# B&R Automation Studio project HISTest (part 6)

#### PMSDataTxParsing.st
```iecst
ACTION ActPMSDATATxParshing:

	PMS.SysBatProduct.Value[0]		:= SHL(USINT_TO_DWORD(PMS.SysBatProduct.Field.BSA_Production_Num), 24) OR SHL(USINT_TO_DWORD(PMS.SysBatProduct.Field.BSA_Production_Type), 16) OR UINT_TO_DWORD(PMS.SysBatProduct.Field.BSA_Production_Year);
	PMS.SysBatProduct.Value[1]		:= SHL(USINT_TO_DWORD(PMS.SysBatProduct.Field.BSA_Production_BSA_Parallel), 16) OR SHL(USINT_TO_DWORD(PMS.SysBatProduct.Field.BSA_Production_BSA_Serial), 8) OR USINT_TO_DWORD(PMS.SysBatProduct.Field.BSA_Production_VER);

	PMS.SysBatCal.Value[0]			:= SHL(REAL_TO_DWORD(PMS.SysBatCal.Field.BSA_Curr_Total), 16) OR REAL_TO_DWORD(PMS.SysBatCal.Field.BSA_Volt_Total);
	PMS.SysBatCal.Value[1] 			:= SHL(UINT_TO_DWORD(PMS.SysBatCal.Field.BSA_Divice_Status), 16) OR REAL_TO_DWORD(PMS.SysBatCal.Field.BSA_SOC);

	PMS.SysBatPWR.Value[0]			:= SHL(REAL_TO_DWORD(PMS.SysBatPWR.Field.BSA_Peak_Charge_Power_Limit), 16) OR REAL_TO_DWORD(PMS.SysBatPWR.Field.BSA_Cont_Charge_Power_Limit);
	PMS.SysBatPWR.Value[1] 			:= SHL(REAL_TO_DWORD(PMS.SysBatPWR.Field.BSA_Peak_Discharge_Power_Limit), 16) OR REAL_TO_DWORD(PMS.SysBatPWR.Field.BSA_Cont_Discharge_Power_Limit);

	PMS.SysCellVolt.Value[0]		:= SHL(REAL_TO_DWORD(PMS.SysCellVolt.Field.BSA_Cell_MinV), 16) OR REAL_TO_DWORD(PMS.SysCellVolt.Field.BSA_Cell_MaxV);
	PMS.SysCellVolt.Value[1] 		:= SHL(REAL_TO_DWORD(PMS.SysCellVolt.Field.BSA_Cell_DeviV), 16) OR REAL_TO_DWORD(PMS.SysCellVolt.Field.BSA_Cell_AVGV);

	PMS.SysCellTemps.Value[0]		:= SHL(REAL_TO_DWORD(PMS.SysCellTemps.Field.BSA_Cell_MinT), 16) OR REAL_TO_DWORD(PMS.SysCellTemps.Field.BSA_Cell_MaxT);
	PMS.SysCellTemps.Value[1] 		:= SHL(REAL_TO_DWORD(PMS.SysCellTemps.Field.BSA_Cell_DeviT), 16) OR REAL_TO_DWORD(PMS.SysCellTemps.Field.BSA_Cell_AVGT);

	PMS.SysCellV_TPos.Value[0]		:= SHL(UINT_TO_DWORD(PMS.SysCellV_TPos.Field.BSA_Cell_MinV_Location), 24) OR SHL(UINT_TO_DWORD(PMS.SysCellV_TPos.Field.BSA_Rack_MinV_Location), 16) OR SHL(USINT_TO_DWORD(PMS.SysCellV_TPos.Field.BSA_Cell_MinV_Location), 8) OR UINT_TO_DWORD(PMS.SysCellV_TPos.Field.BSA_Rack_MaxV_Location);
	PMS.SysCellV_TPos.Value[1] 		:= SHL(UINT_TO_DWORD(PMS.SysCellV_TPos.Field.BSA_Cell_MinT_Location), 24) OR SHL(UINT_TO_DWORD(PMS.SysCellV_TPos.Field.BSA_Rack_MinT_Location), 16) OR SHL(USINT_TO_DWORD(PMS.SysCellV_TPos.Field.BSA_Cell_MinT_Location), 8) OR UINT_TO_DWORD(PMS.SysCellV_TPos.Field.BSA_Rack_MaxT_Location);

	PMS.SysBatProtect.Value[0].0	:=	PMS.SysBatProtect.Field.BSA_Alarm_OC	;
	PMS.SysBatProtect.Value[0].1	:=	PMS.SysBatProtect.Field.BSA_Alarm_SOC_OV	;
	PMS.SysBatProtect.Value[0].2	:=	PMS.SysBatProtect.Field.BSA_Alarm_SOC_UN	;
	PMS.SysBatProtect.Value[0].3	:=	PMS.SysBatProtect.Field.BSA_Alarm_OV	;
	PMS.SysBatProtect.Value[0].4	:=	PMS.SysBatProtect.Field.BSA_Alarm_UV	;
	PMS.SysBatProtect.Value[0].5	:=	PMS.SysBatProtect.Field.BSA_Alarm_Cell_OV	;
	PMS.SysBatProtect.Value[0].6	:=	PMS.SysBatProtect.Field.BSA_Alarm_Cell_UV	;
	PMS.SysBatProtect.Value[0].7	:=	PMS.SysBatProtect.Field.BSA_Alarm_Cell_UnBalaV	;
	PMS.SysBatProtect.Value[0].8	:=	PMS.SysBatProtect.Field.BSA_Alarm_Discharger_Cell_OT	;
	PMS.SysBatProtect.Value[0].9	:=	PMS.SysBatProtect.Field.BSA_Alarm_Charger_Cell_OT	;
	PMS.SysBatProtect.Value[0].10	:=	PMS.SysBatProtect.Field.BSA_Alarm_Discharger_Cell_UT	;
	PMS.SysBatProtect.Value[0].11	:=	PMS.SysBatProtect.Field.BSA_Alarm_Charger_Cell_UT	;
	PMS.SysBatProtect.Value[0].12	:=	PMS.SysBatProtect.Field.BSA_Alarm_Cell_UnBalaT	;
	PMS.SysBatProtect.Value[0].13	:=	PMS.SysBatProtect.Field.BSA_Alarm_Continuously_OP	;
	PMS.SysBatProtect.Value[0].14	:=	PMS.SysBatProtect.Field.BSA_Alarm_Peak_OP	;

	PMS.SysBatProtect.Value[0].16	:=	PMS.SysBatProtect.Field.BSA_Fault_OC	;
	PMS.SysBatProtect.Value[0].17	:=	PMS.SysBatProtect.Field.BSA_Fault_SOC_OV	;
	PMS.SysBatProtect.Value[0].18	:=	PMS.SysBatProtect.Field.BSA_Fault_SOC_UN	;
	PMS.SysBatProtect.Value[0].19	:=	PMS.SysBatProtect.Field.BSA_Fault_OV	;
	PMS.SysBatProtect.Value[0].20	:=	PMS.SysBatProtect.Field.BSA_Fault_UV	;
	PMS.SysBatProtect.Value[0].21	:=	PMS.SysBatProtect.Field.BSA_Fault_Cell_OV	;
	PMS.SysBatProtect.Value[0].22	:=	PMS.SysBatProtect.Field.BSA_Fault_Cell_UV	;
	PMS.SysBatProtect.Value[0].23	:=	PMS.SysBatProtect.Field.BSA_Fault_Cell_UnBalaV	;
	PMS.SysBatProtect.Value[0].24	:=	PMS.SysBatProtect.Field.BSA_Fault_Discharger_Cell_OT	;
	PMS.SysBatProtect.Value[0].25	:=	PMS.SysBatProtect.Field.BSA_Fault_Charger_Cell_OT	;
	PMS.SysBatProtect.Value[0].26	:=	PMS.SysBatProtect.Field.BSA_Fault_Discharger_Cell_UT	;
	PMS.SysBatProtect.Value[0].27	:=	PMS.SysBatProtect.Field.BSA_Fault_Charger_Cell_UT	;
	PMS.SysBatProtect.Value[0].28	:=	PMS.SysBatProtect.Field.BSA_Fault_Cell_UnBalaT	;
	PMS.SysBatProtect.Value[0].29	:=	PMS.SysBatProtect.Field.BSA_Fault_Continuously_OP	;
	PMS.SysBatProtect.Value[0].30	:=	PMS.SysBatProtect.Field.BSA_Fault_Peak_OP	;
	PMS.SysBatProtect.Value[1].0	:=	PMS.SysBatProtect.Field.BSA_Prtct_OC	;
	PMS.SysBatProtect.Value[1].1	:=	PMS.SysBatProtect.Field.BSA_Prtct_SOC_OV	;
	PMS.SysBatProtect.Value[1].2	:=	PMS.SysBatProtect.Field.BSA_Prtct_SOC_UN	;
	PMS.SysBatProtect.Value[1].3	:=	PMS.SysBatProtect.Field.BSA_Prtct_OV	;
	PMS.SysBatProtect.Value[1].4	:=	PMS.SysBatProtect.Field.BSA_Prtct_UV	;
	PMS.SysBatProtect.Value[1].5	:=	PMS.SysBatProtect.Field.BSA_Prtct_Cell_OV	;
	PMS.SysBatProtect.Value[1].6	:=	PMS.SysBatProtect.Field.BSA_Prtct_Cell_UV	;
	PMS.SysBatProtect.Value[1].7	:=	PMS.SysBatProtect.Field.BSA_Prtct_Cell_UnBalaV	;
	PMS.SysBatProtect.Value[1].8	:=	PMS.SysBatProtect.Field.BSA_Prtct_Discharger_Cell_OT	;
	PMS.SysBatProtect.Value[1].9	:=	PMS.SysBatProtect.Field.BSA_Prtct_Charger_Cell_OT	;
	PMS.SysBatProtect.Value[1].10	:=	PMS.SysBatProtect.Field.BSA_Prtct_Discharger_Cell_UT	;
	PMS.SysBatProtect.Value[1].11	:=	PMS.SysBatProtect.Field.BSA_Prtct_Charger_Cell_UT	;
	PMS.SysBatProtect.Value[1].12	:=	PMS.SysBatProtect.Field.BSA_Prtct_Cell_UnBalaT	;
	PMS.SysBatProtect.Value[1].13	:=	PMS.SysBatProtect.Field.BSA_Prtct_Continuously_OP	;
	PMS.SysBatProtect.Value[1].14	:=	PMS.SysBatProtect.Field.BSA_Prtct_Peak_OP	;
	PMS.SysBatProtect.Value[1].15	:=	PMS.SysBatProtect.Field.BSA_Prtct_InternalCOM	;
	PMS.SysBatProtect.Value[1].16	:=	PMS.SysBatProtect.Field.BSA_Prtct_ExternalCOM	;
	PMS.SysBatProtect.Value[1].17	:=	PMS.SysBatProtect.Field.BSA_Prtct_RelayWelding	;
	PMS.SysBatProtect.Value[1].18	:=	PMS.SysBatProtect.Field.BSA_Prtct_WaterLeak	;
	PMS.SysBatProtect.Value[1].19	:=	PMS.SysBatProtect.Field.BSA_Prtct_InsulationReg	;
	PMS.SysBatProtect.Value[1].20	:=	PMS.SysBatProtect.Field.BSA_Prtct_MDSFuse	;
	PMS.SysBatProtect.Value[1].21	:=	PMS.SysBatProtect.Field.BSA_Prtct_Cooling_System	;

	PMS.SysBatDIO.Value[0].0		:=	PMS.SysBatDIO.Field.BSA_Prelay_DO_Status	;
	PMS.SysBatDIO.Value[0].1		:=	PMS.SysBatDIO.Field.BSA_Nrelay_DO_Status	;
	PMS.SysBatDIO.Value[0].2		:=	PMS.SysBatDIO.Field.BSA_ProRelay_DO_Status	;
	PMS.SysBatDIO.Value[0].3		:=	PMS.SysBatDIO.Field.BSA_Buzzer_DO_Status	;
	PMS.SysBatDIO.Value[0].4		:=	PMS.SysBatDIO.Field.BSA_PowerLamp_DO_Status	;
	PMS.SysBatDIO.Value[0].5		:=	PMS.SysBatDIO.Field.BSA_DO_Spare06	;
	PMS.SysBatDIO.Value[0].6		:=	PMS.SysBatDIO.Field.BSA_DO_Spare07	;
	PMS.SysBatDIO.Value[0].7		:=	PMS.SysBatDIO.Field.BSA_DO_Spare08	;
	PMS.SysBatDIO.Value[0].8		:=	PMS.SysBatDIO.Field.BSA_DO_Spare09	;
	PMS.SysBatDIO.Value[0].9		:=	PMS.SysBatDIO.Field.BSA_DO_Spare10	;
	PMS.SysBatDIO.Value[0].10		:=	PMS.SysBatDIO.Field.BSA_DO_Spare11	;
	PMS.SysBatDIO.Value[0].11		:=	PMS.SysBatDIO.Field.BSA_DO_Spare12	;
	PMS.SysBatDIO.Value[0].12		:=	PMS.SysBatDIO.Field.BSA_PRelayAUX_DI_Status	;
	PMS.SysBatDIO.Value[0].13		:=	PMS.SysBatDIO.Field.BSA_NRelayAUX_DI_Status	;
	PMS.SysBatDIO.Value[0].14		:=	PMS.SysBatDIO.Field.BSA_EMGSwitch_DI_Status ;
	PMS.SysBatDIO.Value[0].15		:=	PMS.SysBatDIO.Field.BSA_CoolingSystem_DI_Status  ;
	PMS.SysBatDIO.Value[0].16		:=	PMS.SysBatDIO.Field.BSA_MDS_DI_Status	;
	PMS.SysBatDIO.Value[0].17		:=	PMS.SysBatDIO.Field.BSA_DI_Spare06	;
	PMS.SysBatDIO.Value[0].18		:=	PMS.SysBatDIO.Field.BSA_DI_Spare07	;
	PMS.SysBatDIO.Value[0].19		:=	PMS.SysBatDIO.Field.BSA_DI_Spare08	;
	PMS.SysBatDIO.Value[0].20		:=	PMS.SysBatDIO.Field.BSA_DI_Spare09	;
	PMS.SysBatDIO.Value[0].21		:=	PMS.SysBatDIO.Field.BSA_DI_Spare10	;
	PMS.SysBatDIO.Value[0].22		:=	PMS.SysBatDIO.Field.BSA_DI_Spare11	;
	PMS.SysBatDIO.Value[0].23		:=	PMS.SysBatDIO.Field.BSA_DI_Spare12	;
	PMS.SysBatDIO.Value[1]			:= SHL(REAL_TO_DWORD(PMS.SysBatDIO.Field.BSA_SOH), 16);

	PMS.BRACal.Value[0]				:= SHL(REAL_TO_DWORD(PMS.BRACal.Field.BRA_Volt_Total), 16) OR UINT_TO_DWORD(PMS.BRACal.Field.BRA_Rack_Num);
	PMS.BRACal.Value[1] 			:= SHL(REAL_TO_DWORD(PMS.BRACal.Field.BRA_SOC), 16) OR REAL_TO_DWORD(PMS.BRACal.Field.BRA_Curr_Total);

	PMS.BRAPWR_A.Value[0]			:= SHL(REAL_TO_DWORD(PMS.BRAPWR_A.Field.BRA_SOH), 16) OR UINT_TO_DWORD(PMS.BRAPWR_A.Field.BRA_Rack_Num);
	PMS.BRAPWR_A.Value[1] 			:= SHL(REAL_TO_DWORD(PMS.BRAPWR_A.Field.BRA_Peak_CHA_PWR_Limit), 16) OR REAL_TO_DWORD(PMS.BRAPWR_A.Field.BRA_CONT_CHA_PWR_Limit);

	PMS.BRAPWR_B.Value[0]			:= SHL(REAL_TO_DWORD(PMS.BRAPWR_B.Field.BRA_CONT_DisCHA_PWR_Limit), 16) OR UINT_TO_DWORD(PMS.BRACal.Field.BRA_Rack_Num);
	PMS.BRAPWR_B.Value[1] 			:= REAL_TO_DWORD(PMS.BRAPWR_B.Field.BRA_Peak_DisCHA_PWR_Limit);

	PMS.BRACal.Value[0]				:= SHL(REAL_TO_DWORD(PMS.BRACal.Field.BRA_Volt_Total), 16) OR UINT_TO_DWORD(PMS.BRACal.Field.BRA_Rack_Num);
	PMS.BRACal.Value[1] 			:= SHL(REAL_TO_DWORD(PMS.BRACal.Field.BRA_SOC), 16) OR REAL_TO_DWORD(PMS.BRACal.Field.BRA_Curr_Total);

	PMS.BRACellV.Value[0]			:= SHL(REAL_TO_DWORD(PMS.BRACellV.Field.BRA_Cell_Max_Voltage), 16) OR UINT_TO_DWORD(PMS.BRACellV.Field.BRA_Rack_Num);
	PMS.BRACellV.Value[1] 			:= SHL(REAL_TO_DWORD(PMS.BRACellV.Field.BRA_Cell_AGV_Voltage), 16) OR REAL_TO_DWORD(PMS.BRACellV.Field.BRA_Cell_Min_Voltage);

	PMS.BRACellT.Value[0]			:= SHL(REAL_TO_DWORD(PMS.BRACellT.Field.BRA_Cell_Max_Temperature), 16) OR REAL_TO_DWORD(PMS.BRACellT.Field.BRA_Rack_Num);
	PMS.BRACellT.Value[1] 			:= SHL(REAL_TO_DWORD(PMS.BRACellT.Field.BRA_Cell_AGV_Temperature), 16) OR REAL_TO_DWORD(PMS.BRACellT.Field.BRA_Cell_Min_Temperature);

	PMS.BRACellDiv.Value[0]			:= SHL(REAL_TO_DWORD(PMS.BRACellDiv.Field.BRA_Cell_DIV_Voltage), 16) OR UINT_TO_DWORD(PMS.BRACellDiv.Field.BRA_Rack_Num);
	PMS.BRACellDiv.Value[1] 		:= REAL_TO_DWORD(PMS.BRACellDiv.Field.BRA_Cell_DIV_Temperature);

	PMS.BRA_VTPos.Value[0]			:= SHL(USINT_TO_DWORD(PMS.BRA_VTPos.Field.BRA_Min_Cell_V_Location), 24) OR SHL(USINT_TO_DWORD(PMS.BRA_VTPos.Field.BRA_Max_Cell_V_Location), 16) OR UINT_TO_DWORD(PMS.BRA_VTPos.Field.BRA_Rack_Num);
	PMS.BRA_VTPos.Value[1] 			:= SHL(USINT_TO_DWORD(PMS.BRA_VTPos.Field.BRA_Min_Cell_T_Location), 8) OR USINT_TO_DWORD(PMS.BRA_VTPos.Field.BRA_Max_Cell_V_Location);

	PMS.BAR_Alarm.Value[0]			:= UINT_TO_DWORD(PMS.BAR_Alarm.Field.BRA_Rack_Num);
	PMS.BAR_Alarm.Value[0].16		:=	PMS.BAR_Alarm.Field.BRA_Alarm_OC	;
	PMS.BAR_Alarm.Value[0].17		:=	PMS.BAR_Alarm.Field.BRA_Alarm_SOC_OV	;
	PMS.BAR_Alarm.Value[0].18		:=	PMS.BAR_Alarm.Field.BRA_Alarm_SOC_UN	;
	PMS.BAR_Alarm.Value[0].19		:=	PMS.BAR_Alarm.Field.BRA_Alarm_OV	;
	PMS.BAR_Alarm.Value[0].20		:=	PMS.BAR_Alarm.Field.BRA_Alarm_UV	;
	PMS.BAR_Alarm.Value[0].21		:=	PMS.BAR_Alarm.Field.BRA_Alarm_Cell_OV	;
	PMS.BAR_Alarm.Value[0].22		:=	PMS.BAR_Alarm.Field.BRA_Alarm_Cell_UV	;
	PMS.BAR_Alarm.Value[0].23		:=	PMS.BAR_Alarm.Field.BRA_Alarm_Cell_UnBalaV	;
	PMS.BAR_Alarm.Value[0].24		:=	PMS.BAR_Alarm.Field.BRA_Alarm_Discharger_Cell_OT	;
	PMS.BAR_Alarm.Value[0].25		:=	PMS.BAR_Alarm.Field.BRA_Alarm_Charger_Cell_OT	;
	PMS.BAR_Alarm.Value[0].26		:=	PMS.BAR_Alarm.Field.BRA_Alarm_Discharger_Cell_OT	;
	PMS.BAR_Alarm.Value[0].27		:=	PMS.BAR_Alarm.Field.BRA_Alarm_Charger_Cell_UT	;
	PMS.BAR_Alarm.Value[0].28		:=	PMS.BAR_Alarm.Field.BRA_Alarm_Cell_UnBalaT	;
	PMS.BAR_Alarm.Value[0].29		:=	PMS.BAR_Alarm.Field.BRA_Alarm_Continuously_OP	;
	PMS.BAR_Alarm.Value[0].30		:=	PMS.BAR_Alarm.Field.BRA_Alarm_Peak_OP	;
	PMS.BAR_Alarm.Value[1].0		:=	PMS.BAR_Alarm.Field.BRA_Fault_OC	;
	PMS.BAR_Alarm.Value[1].1		:=	PMS.BAR_Alarm.Field.BRA_Fault_SOC_OV	;
	PMS.BAR_Alarm.Value[1].2		:=	PMS.BAR_Alarm.Field.BRA_Fault_SOC_UN	;
	PMS.BAR_Alarm.Value[1].3		:=	PMS.BAR_Alarm.Field.BRA_Fault_OV	;
	PMS.BAR_Alarm.Value[1].4		:=	PMS.BAR_Alarm.Field.BRA_Fault_UV	;
	PMS.BAR_Alarm.Value[1].5		:=	PMS.BAR_Alarm.Field.BRA_Fault_Cell_OV	;
	PMS.BAR_Alarm.Value[1].6		:=	PMS.BAR_Alarm.Field.BRA_Fault_Cell_UV	;
	PMS.BAR_Alarm.Value[1].7		:=	PMS.BAR_Alarm.Field.BRA_Fault_Cell_UnBalaV	;
	PMS.BAR_Alarm.Value[1].8		:=	PMS.BAR_Alarm.Field.BRA_Fault_Discharger_Cell_OT	;
	PMS.BAR_Alarm.Value[1].9		:=	PMS.BAR_Alarm.Field.BRA_Fault_Charger_Cell_OT	;
	PMS.BAR_Alarm.Value[1].10		:=	PMS.BAR_Alarm.Field.BRA_Fault_Discharger_Cell_OT	;
	PMS.BAR_Alarm.Value[1].11		:=	PMS.BAR_Alarm.Field.BRA_Fault_Charger_Cell_UT	;
	PMS.BAR_Alarm.Value[1].12		:=	PMS.BAR_Alarm.Field.BRA_Fault_Cell_UnBalaT	;
	PMS.BAR_Alarm.Value[1].13		:=	PMS.BAR_Alarm.Field.BRA_Fault_Continuously_OP	;
	PMS.BAR_Alarm.Value[1].14		:=	PMS.BAR_Alarm.Field.BRA_Fault_Peak_OP	;

	PMS.BAR_Protect.Value[0]		:= UINT_TO_DWORD(PMS.BAR_Protect.Field.BRA_Rack_Num);
	PMS.BAR_Protect.Value[0].16		:=	PMS.BAR_Protect.Field.BRA_Prtct_OC	;
	PMS.BAR_Protect.Value[0].17		:=	PMS.BAR_Protect.Field.BRA_Prtct_SOC_OV	;
	PMS.BAR_Protect.Value[0].18		:=	PMS.BAR_Protect.Field.BRA_Prtct_SOC_UN	;
	PMS.BAR_Protect.Value[0].19		:=	PMS.BAR_Protect.Field.BRA_Prtct_OV	;
	PMS.BAR_Protect.Value[0].20		:=	PMS.BAR_Protect.Field.BRA_Prtct_UV	;
	PMS.BAR_Protect.Value[0].21		:=	PMS.BAR_Protect.Field.BRA_Prtct_Cell_OV	;
	PMS.BAR_Protect.Value[0].22		:=	PMS.BAR_Protect.Field.BRA_Prtct_Cell_UV	;
	PMS.BAR_Protect.Value[0].23		:=	PMS.BAR_Protect.Field.BRA_Prtct_Cell_UnBalaV	;
	PMS.BAR_Protect.Value[0].24		:=	PMS.BAR_Protect.Field.BRA_Prtct_Discharger_Cell_OT	;
	PMS.BAR_Protect.Value[0].25		:=	PMS.BAR_Protect.Field.BRA_Prtct_Charger_Cell_OT	;
	PMS.BAR_Protect.Value[0].26		:=	PMS.BAR_Protect.Field.BRA_Prtct_Discharger_Cell_UT	;
	PMS.BAR_Protect.Value[0].27		:=	PMS.BAR_Protect.Field.BRA_Prtct_Charger_Cell_UT	;
	PMS.BAR_Protect.Value[0].28		:=	PMS.BAR_Protect.Field.BRA_Prtct_Cell_UnBalaT	;
	PMS.BAR_Protect.Value[0].29		:=	PMS.BAR_Protect.Field.BRA_Prtct_Continuously_OP	;
	PMS.BAR_Protect.Value[0].30		:=	PMS.BAR_Protect.Field.BRA_Prtct_Peak_OP	;
	PMS.BAR_Protect.Value[0].31		:=	PMS.BAR_Protect.Field.BRA_Prtct_InternalCOM	;
	PMS.BAR_Protect.Value[1].0		:=	PMS.BAR_Protect.Field.BRA_Prtct_ExternalCOM	;
	PMS.BAR_Protect.Value[1].1		:=	PMS.BAR_Protect.Field.BRA_Prtct_RelayWelding	;
	PMS.BAR_Protect.Value[1].2		:=	PMS.BAR_Protect.Field.BRA_Prtct_WaterLeak	;
	PMS.BAR_Protect.Value[1].3		:=	PMS.BAR_Protect.Field.BRA_Prtct_InsulationReg	;
	PMS.BAR_Protect.Value[1].4		:=	PMS.BAR_Protect.Field.BRA_Prtct_MDSFuse	;
	PMS.BAR_Protect.Value[1].5		:=	PMS.BAR_Protect.Field.BRA_Prtct_CoolingSystem	;

	PMS.BAR_DIO.Value[0]			:= UINT_TO_DWORD(PMS.BAR_DIO.Field.BRA_Rack_Num);
	PMS.BAR_DIO.Value[0].16			:=	PMS.BAR_DIO.Field.BRA_Prelay_DO_Status 	;
	PMS.BAR_DIO.Value[0].17			:=	PMS.BAR_DIO.Field.BRA_Nrelay_DO_Status	;
	PMS.BAR_DIO.Value[0].18			:=	PMS.BAR_DIO.Field.BRA_ProRelay_DO_Status	;
	PMS.BAR_DIO.Value[0].19			:=	PMS.BAR_DIO.Field.BRA_PowerLamp_DO_Status	;
	PMS.BAR_DIO.Value[0].20			:=	PMS.BAR_DIO.Field.BRA_Buzzer_DO_Status	;
	PMS.BAR_DIO.Value[1].0			:=	PMS.BAR_DIO.Field.BRA_PRelayAUX_DI_Status	;
	PMS.BAR_DIO.Value[1].1			:=	PMS.BAR_DIO.Field.BRA_NRelayAUX_DI_Status	;
	PMS.BAR_DIO.Value[1].2			:=	PMS.BAR_DIO.Field.BRA_EMGSwitch_DI_Status	;
	PMS.BAR_DIO.Value[1].3			:=	PMS.BAR_DIO.Field.BRA_MDS_DI_Status	;

	PMS.BAR_DIO.Value[1].16			:=	PMS.BAR_DIO.Field.BRA_Waterleak_Dete_MD1	;
	PMS.BAR_DIO.Value[1].17			:=	PMS.BAR_DIO.Field.BRA_Waterleak_Dete_MD2	;
	PMS.BAR_DIO.Value[1].18			:=	PMS.BAR_DIO.Field.BRA_Waterleak_Dete_MD3	;
	PMS.BAR_DIO.Value[1].19			:=	PMS.BAR_DIO.Field.BRA_Waterleak_Dete_MD4	;
	PMS.BAR_DIO.Value[1].20			:=	PMS.BAR_DIO.Field.BRA_Waterleak_Dete_MD5	;
	PMS.BAR_DIO.Value[1].21			:=	PMS.BAR_DIO.Field.BRA_Waterleak_Dete_MD6	;
	PMS.BAR_DIO.Value[1].22			:=	PMS.BAR_DIO.Field.BRA_Waterleak_Dete_MD7	;

END_ACTION
```

### Program Logical/Source/PMS_CAN/CANRxPMS (IEC)

#### ArCanReceive.st - Cyclic code
```iecst
PROGRAM _INIT

	ActArCanReceiver;
	ArCanReceiver.enable				:= TRUE;
	ArCanReceiver.receiverDeviceName 	:= 'IF6.ST5.IF1';       (* for X20CS1070 *)
	ArCanReceiver.id					:= 0;
	ArCanReceiver.idMask				:= arCAN_RECEIVE_ALL;  // or configure IDMask
	ArCanReceiver.format				:= arCAN_11BIT;  // or arCAN_29BIT
	ArCanReceiver.queueSize				:= 128;
	ArCanReceiver.ArCanSetBitTimingRegisters_0.Register0 := 0;
	ArCanReceiver.ArCanSetBitTimingRegisters_0.Register1 := 16#1C;

	(**********************	 CAN Baud rate Register Value	*************************)
	(********************************************************************************)
	(* 	  1 000 000 bit/s    >>		Register0 = 16#00	||		Register1 = 16#14	*)
	(* 		800 000 bit/s    >>		Register0 = 16#00	||		Register1 = 16#16	*)
	(* 		500 000 bit/s    >>		Register0 = 16#00	||		Register1 = 16#1C	*)
	(* 		250 000 bit/s    >>		Register0 = 16#01	||		Register1 = 16#1C	*)
	(* 		125 000 bit/s    >>		Register0 = 16#03	||		Register1 = 16#1C	*)
	(* 		100 000 bit/s    >>		Register0 = 16#04	||		Register1 = 16#1C	*)
	(* 		050 000 bit/s    >>		Register0 = 16#09	||		Register1 = 16#1C	*)
	(* 		020 000 bit/s    >>		Register0 = 16#18	||		Register1 = 16#1C	*)
	(* 		010 000 bit/s    >>		Register0 = 16#31	||		Register1 = 16#1C	*)
	(********************************************************************************)
	(********************************************************************************)

END_PROGRAM

PROGRAM _CYCLIC

	(* Action for ArCanReceiver *)
	ActArCanReceiver;
	(***********************************************************)
	(* Customize the received data *)
	// ArCanReceiver.ArCanReceiver_0.ReceivedFrame; //Data received
	IF (ArCanReceiver.ArCanReceiver_0.NewDataValid) THEN

		CASE ArCanReceiver.ArCanReceiver_0.ReceivedFrame.ID OF

			16#700: // PMS

			IF ArCanReceiver.ArCanReceiver_0.ReceivedFrame.ID = 16#700 THEN
				memcpy(ADR(PMS.PMS.Value), ADR(ArCanReceiver.ArCanReceiver_0.ReceivedFrame.Data), SIZEOF(PMS.PMS.Value));
			END_IF;

		END_CASE;

	END_IF

	ActPMSDATARxParshing;

	(***********************************************************)
	(* CAN Communication Status *)
	(***********************************************************)

	IF ArCanReceiver.ArCanReceiver_0.Error THEN
		gComm.CAN1.bError	:= TRUE;
		gComm.CAN1.bActive	:= FALSE;
		gComm.CAN1.bTransmitting	:= FALSE;
	ELSIF ArCanReceiver.ArCanReceiver_0.Active AND ArCanReceiver.ArCanReceiver_0.Busy THEN
		gComm.CAN1.bError	:= FALSE;
		gComm.CAN1.bActive	:= TRUE;

		IF (countCANSuccessOld <> ArCanReceiver.successCount) THEN
			countCANSuccessOld	:= ArCanReceiver.successCount;
			gComm.CAN1.bTransmitting	:= TRUE;
			countTime	:= 0;
		ELSE
			countTime	:= countTime + 1;
			IF (countTime > 50) THEN
				gComm.CAN1.bTransmitting	:= FALSE;
				countTime	:= 0;
			END_IF
		END_IF
	ELSE
		gComm.CAN1.bError	:= FALSE;
		gComm.CAN1.bActive	:= FALSE;
		gComm.CAN1.bTransmitting	:= FALSE;
	END_IF
	(***********************************************************)

END_PROGRAM

PROGRAM _EXIT

	(* Deinitialization of the receiver *)
	ArCanReceiver.ArCanReceiver_0.Enable	:= FALSE;
	ArCanReceiver.ArCanReceiver_0();

END_PROGRAM
```

#### PMSDataRxParsing.st
```iecst
ACTION ActPMSDATARxParshing:

	PMS.PMS.Field.PMS_WakeUp_CMD							:=	PMS.PMS.Value[0].0;
	PMS.PMS.Field.PMS_POWER_CMD								:=	PMS.PMS.Value[0].1;
	PMS.PMS.Field.PMS_FaultReset							:=	PMS.PMS.Value[0].8;
	PMS.PMS.Field.PMS_Po_RelayStatus						:=	PMS.PMS.Value[0].16;
	PMS.PMS.Field.PMS_Pro_RelayStatus						:=	PMS.PMS.Value[0].17;
	PMS.PMS.Field.PMS_Ne_RelayStatus						:=	PMS.PMS.Value[0].18;

END_ACTION
```

### Program Logical/Source/PMS_CAN/PMSRxHandle (IEC)

#### Main.st
```iecst
PROGRAM _INIT
	(* Insert code here *)

END_PROGRAM

PROGRAM _CYCLIC
	(* Insert code here *)

	Sys.WakeUpSig := PMS.PMS.Field.PMS_WakeUp_CMD;

END_PROGRAM

PROGRAM _EXIT
	(* Insert code here *)

END_PROGRAM
```

### Program Logical/Source/PMS_CAN/PMS_Calculator (IEC)

#### Main.st - Init, cyclic, exit code
```iecst
PROGRAM _INIT
	(* Insert code here *)

END_PROGRAM

PROGRAM _CYCLIC
	(* Insert code here *)

	SubBMS_Calculator.BSA[0] := SubBMS.Rack1.BSA;
	SubBMS_Calculator.BSA[1] := SubBMS.Rack2.BSA;
	SubBMS_Calculator.BSA[2] := SubBMS.Rack3.BSA;
	SubBMS_Calculator.BSA[3] := SubBMS.Rack4.BSA;

	SubBMS.Rack1.BMA.Field := SubBMS_Calculator.BMA[0].Field;
	SubBMS.Rack2.BMA.Field := SubBMS_Calculator.BMA[1].Field;
	SubBMS.Rack3.BMA.Field := SubBMS_Calculator.BMA[2].Field;
	SubBMS.Rack4.BMA.Field := SubBMS_Calculator.BMA[3].Field;

	PMS_SysBatCal;
	PMS_SysBatPWR;
	PMS_SysCell_Volt_Location;
	PMS_SysCell_Temps_Location;
	PMS_SysBatProtect;
	PMS_SysBatDIO;
	PMS_BRACal;
	PMS_BRAPWR_A;
	PMS_BRAPWR_B;
	PMS_BRACellV;
	PMS_BRACellT;
	PMS_BRACellDiv;
	PMS_BRA_VTPos;
	PMS_BAR_Alarm;
	PMS_BAR_Protect;
	PMS_BAR_DIO;

	System_RackState;
	System_RackVolt;
	System_RackCurr;
	System_RackTotal;
END_PROGRAM

PROGRAM _EXIT
	(* Insert code here *)

END_PROGRAM
```

#### Variables.var - Local variables
```iecst
VAR
	LoopCount : USINT;
END_VAR
```

#### PMS_Calculator.st
```iecst
ACTION PMS_SysBatCal:

	PMS.SysBatCal.Field.BSA_Volt_Total := -32767;
	PMS.SysBatCal.Field.BSA_Curr_Total := 0;
	PMS.SysBatCal.Field.BSA_SOC := 0;
	PMS.SysBatDIO.Field.BSA_SOH := 0;

	FOR LoopCount := 0 TO RACK_MAXNUM_MINUS_1 DO

		IF HMI.RackEnable[LoopCount] THEN
			PMS.SysBatCal.Field.BSA_Curr_Total 	:= PMS.SysBatCal.Field.BSA_Curr_Total + SubBMS_Calculator.BSA[LoopCount].Rack_Calc.Field.BRA_Curr_Total;
			PMS.SysBatCal.Field.BSA_SOC 		:= PMS.SysBatCal.Field.BSA_SOC + SubBMS_Calculator.BSA[LoopCount].Rack_Calc.Field.BRA_SOC;
			PMS.SysBatDIO.Field.BSA_SOH 		:= PMS.SysBatDIO.Field.BSA_SOH + SubBMS_Calculator.BSA[LoopCount].Rack_Calc.Field.BRA_SOH;

			IF SubBMS_Calculator.BSA[LoopCount].Rack_Calc.Field.BRA_Volt_Total > PMS.SysBatCal.Field.BSA_Volt_Total THEN
				PMS.SysBatCal.Field.BSA_Volt_Total := SubBMS_Calculator.BSA[LoopCount].Rack_Calc.Field.BRA_Volt_Total;
			END_IF;
		END_IF;
	END_FOR;

END_ACTION

ACTION PMS_SysBatPWR:
	PMS.SysBatPWR.Field.BSA_Cont_Charge_Power_Limit := -32767;
	PMS.SysBatPWR.Field.BSA_Peak_Charge_Power_Limit := -32767;
	PMS.SysBatPWR.Field.BSA_Cont_Discharge_Power_Limit := -32767;
	PMS.SysBatPWR.Field.BSA_Peak_Discharge_Power_Limit := -32767;

	FOR LoopCount := 0 TO RACK_MAXNUM_MINUS_1 DO

		IF HMI.RackEnable[LoopCount] THEN
			IF SubBMS_Calculator.BSA[LoopCount].Rack_PWRCalc.Field.BSA_CHAPWCont > PMS.SysBatPWR.Field.BSA_Cont_Charge_Power_Limit THEN
				PMS.SysBatPWR.Field.BSA_Cont_Charge_Power_Limit 		:= SubBMS_Calculator.BSA[LoopCount].Rack_PWRCalc.Field.BSA_CHAPWCont;
			END_IF;
			IF SubBMS_Calculator.BSA[LoopCount].Rack_PWRCalc.Field.BSA_DisCHAPWCont > PMS.SysBatPWR.Field.BSA_Cont_Discharge_Power_Limit THEN
				PMS.SysBatPWR.Field.BSA_Cont_Discharge_Power_Limit 		:= SubBMS_Calculator.BSA[LoopCount].Rack_PWRCalc.Field.BSA_DisCHAPWCont;
			END_IF;
			IF SubBMS_Calculator.BSA[LoopCount].Rack_PWRCalc.Field.BSA_CHAPWPeak > PMS.SysBatPWR.Field.BSA_Peak_Charge_Power_Limit THEN
				PMS.SysBatPWR.Field.BSA_Peak_Charge_Power_Limit 		:= SubBMS_Calculator.BSA[LoopCount].Rack_PWRCalc.Field.BSA_CHAPWPeak;
			END_IF;
			IF SubBMS_Calculator.BSA[LoopCount].Rack_PWRCalc.Field.BSA_DisCHAPWPeak > PMS.SysBatPWR.Field.BSA_Peak_Discharge_Power_Limit THEN
				PMS.SysBatPWR.Field.BSA_Peak_Discharge_Power_Limit 		:= SubBMS_Calculator.BSA[LoopCount].Rack_PWRCalc.Field.BSA_DisCHAPWPeak;
			END_IF;

		END_IF;
	END_FOR;

END_ACTION

ACTION PMS_SysCell_Volt_Location:

	PMS.SysCellVolt.Field.BSA_Cell_MaxV := -32767;
	PMS.SysCellVolt.Field.BSA_Cell_MinV := 32767;

	FOR LoopCount := 0 TO RACK_MAXNUM_MINUS_1 DO

		IF HMI.RackEnable[LoopCount] THEN
			IF SubBMS_Calculator.BSA[LoopCount].Rack_Cell_Vcalc.Field.BSA_Cell_MaxV > PMS.SysCellVolt.Field.BSA_Cell_MaxV THEN

				PMS.SysCellVolt.Field.BSA_Cell_MaxV 			:= SubBMS_Calculator.BSA[LoopCount].Rack_Cell_Vcalc.Field.BSA_Cell_MaxV;

				PMS.SysCellV_TPos.Field.BSA_Rack_MaxV_Location	:= LoopCount + 1;
				PMS.SysCellV_TPos.Field.BSA_Cell_MaxV_Location 	:= UINT_TO_USINT(SubBMS_Calculator.BSA[LoopCount].Rack_Cell_Pcalc.Field.BSA_Cell_MaxV_Location);
			END_IF;

			IF SubBMS_Calculator.BSA[LoopCount].Rack_Cell_Vcalc.Field.BSA_Cell_MinV < PMS.SysCellVolt.Field.BSA_Cell_MinV  THEN

				PMS.SysCellVolt.Field.BSA_Cell_MinV  			:= SubBMS_Calculator.BSA[LoopCount].Rack_Cell_Vcalc.Field.BSA_Cell_MinV;

				PMS.SysCellV_TPos.Field.BSA_Rack_MinV_Location	:= LoopCount + 1;
				PMS.SysCellV_TPos.Field.BSA_Cell_MinV_Location 	:= UINT_TO_USINT(SubBMS_Calculator.BSA[LoopCount].Rack_Cell_Pcalc.Field.BSA_Cell_MinV_Location);
			END_IF;

		END_IF;
	END_FOR;

	PMS.SysCellVolt.Field.BSA_Cell_AVGV 					:= (PMS.SysCellVolt.Field.BSA_Cell_MaxV + PMS.SysCellVolt.Field.BSA_Cell_MinV) / 2;
	PMS.SysCellVolt.Field.BSA_Cell_DeviV 					:= PMS.SysCellVolt.Field.BSA_Cell_MaxV - PMS.SysCellVolt.Field.BSA_Cell_MinV;

END_ACTION

ACTION PMS_SysCell_Temps_Location:

	PMS.SysCellTemps.Field.BSA_Cell_MaxT := -32767;
	PMS.SysCellTemps.Field.BSA_Cell_MinT := 32767;

	FOR LoopCount := 0 TO RACK_MAXNUM_MINUS_1 DO

		IF HMI.RackEnable[LoopCount] THEN
			IF SubBMS_Calculator.BSA[LoopCount].Rack_Cell_Tcalc.Field.BSA_Cell_MaxT > PMS.SysCellTemps.Field.BSA_Cell_MaxT THEN

				PMS.SysCellTemps.Field.BSA_Cell_MaxT 			:= SubBMS_Calculator.BSA[LoopCount].Rack_Cell_Tcalc.Field.BSA_Cell_MaxT;

				PMS.SysCellV_TPos.Field.BSA_Rack_MaxT_Location	:= LoopCount + 1;
				PMS.SysCellV_TPos.Field.BSA_Cell_MaxT_Location 	:= UINT_TO_USINT(SubBMS_Calculator.BSA[LoopCount].Rack_Cell_Pcalc.Field.BSA_Cell_MaxT_Location);
			END_IF;

			IF SubBMS_Calculator.BSA[LoopCount].Rack_Cell_Tcalc.Field.BSA_Cell_MinT < PMS.SysCellTemps.Field.BSA_Cell_MinT  THEN

				PMS.SysCellTemps.Field.BSA_Cell_MinT  			:= SubBMS_Calculator.BSA[LoopCount].Rack_Cell_Tcalc.Field.BSA_Cell_MinT;

				PMS.SysCellV_TPos.Field.BSA_Rack_MinT_Location	:= LoopCount + 1;
				PMS.SysCellV_TPos.Field.BSA_Cell_MinT_Location 	:= UINT_TO_USINT(SubBMS_Calculator.BSA[LoopCount].Rack_Cell_Pcalc.Field.BSA_Cell_MinT_Location);
			END_IF;

		END_IF;
	END_FOR;

	PMS.SysCellTemps.Field.BSA_Cell_AVGT 					:= (PMS.SysCellTemps.Field.BSA_Cell_MaxT + PMS.SysCellTemps.Field.BSA_Cell_MinT) / 2;
	PMS.SysCellTemps.Field.BSA_Cell_DeviT 					:= PMS.SysCellTemps.Field.BSA_Cell_MaxT - PMS.SysCellTemps.Field.BSA_Cell_MinT;

END_ACTION

ACTION PMS_SysBatProtect:
	FOR LoopCount := 0 TO RACK_MAXNUM_MINUS_1 DO
		IF 	SubBMS_Calculator.BSA[LoopCount].Rack_AlarmState.Field.protect.BSA_Prtct_Dischager_OC OR SubBMS_Calculator.BSA[LoopCount].Rack_AlarmState.Field.protect.BSA_Prtct_Chager_OC THEN

			PMS.SysBatProtect.Field.BSA_Prtct_OC := TRUE;

		ELSIF SubBMS_Calculator.BSA[LoopCount].Rack_AlarmState.Field.fault.BSA_FLT_Dischager_OC OR	SubBMS_Calculator.BSA[LoopCount].Rack_AlarmState.Field.fault.BSA_FLT_Chager_OC THEN

			PMS.SysBatProtect.Field.BSA_Fault_OC := TRUE;

		ELSIF SubBMS_Calculator.BSA[LoopCount].Rack_AlarmState.Field.warning.BSA_Wn_Dischager_OC OR	SubBMS_Calculator.BSA[LoopCount].Rack_AlarmState.Field.warning.BSA_Wn_Chager_OC THEN

			PMS.SysBatProtect.Field.BSA_Alarm_OC := TRUE;
		END_IF;

		IF 	SubBMS_Calculator.BSA[LoopCount].Rack_AlarmState.Field.protect.BSA_Prtct_SOC_OV THEN

			PMS.SysBatProtect.Field.BSA_Prtct_SOC_OV  := TRUE;

		ELSIF SubBMS_Calculator.BSA[LoopCount].Rack_AlarmState.Field.fault.BSA_FLT_SOC_OV THEN

			PMS.SysBatProtect.Field.BSA_Fault_SOC_OV  := TRUE;

		ELSIF SubBMS_Calculator.BSA[LoopCount].Rack_AlarmState.Field.warning.BSA_Wn_SOC_OV THEN

			PMS.SysBatProtect.Field.BSA_Alarm_SOC_OV  := TRUE;

		END_IF;

		IF 	SubBMS_Calculator.BSA[LoopCount].Rack_AlarmState.Field.protect.BSA_Prtct_SOC_Un THEN

			PMS.SysBatProtect.Field.BSA_Prtct_SOC_UN  := TRUE;

		ELSIF SubBMS_Calculator.BSA[LoopCount].Rack_AlarmState.Field.fault.BSA_FLT_SOC_Un THEN

			PMS.SysBatProtect.Field.BSA_Fault_SOC_UN  := TRUE;

		ELSIF SubBMS_Calculator.BSA[LoopCount].Rack_AlarmState.Field.warning.BSA_Wn_SOC_Un THEN

			PMS.SysBatProtect.Field.BSA_Alarm_SOC_UN  := TRUE;

		END_IF;

		IF 	SubBMS_Calculator.BSA[LoopCount].Rack_AlarmState.Field.protect.BSA_Prtct_OV THEN

			PMS.SysBatProtect.Field.BSA_Prtct_OV  := TRUE;

		ELSIF SubBMS_Calculator.BSA[LoopCount].Rack_AlarmState.Field.fault.BSA_FLT_OV THEN

			PMS.SysBatProtect.Field.BSA_Fault_OV  := TRUE;

		ELSIF SubBMS_Calculator.BSA[LoopCount].Rack_AlarmState.Field.warning.BSA_Wn_OV THEN

			PMS.SysBatProtect.Field.BSA_Alarm_OV  := TRUE;

		END_IF;

		IF 	SubBMS_Calculator.BSA[LoopCount].Rack_AlarmState.Field.protect.BSA_Prtct_UV THEN

			PMS.SysBatProtect.Field.BSA_Prtct_UV  := TRUE;

		ELSIF SubBMS_Calculator.BSA[LoopCount].Rack_AlarmState.Field.fault.BSA_FLT_UV THEN

			PMS.SysBatProtect.Field.BSA_Fault_UV  := TRUE;

		ELSIF SubBMS_Calculator.BSA[LoopCount].Rack_AlarmState.Field.warning.BSA_Wn_UV THEN

			PMS.SysBatProtect.Field.BSA_Alarm_UV  := TRUE;

		END_IF;

		IF 	SubBMS_Calculator.BSA[LoopCount].Rack_AlarmState.Field.protect.BSA_Prtct_Cell_OV THEN

			PMS.SysBatProtect.Field.BSA_Prtct_Cell_OV  := TRUE;

		ELSIF SubBMS_Calculator.BSA[LoopCount].Rack_AlarmState.Field.fault.BSA_FLT_Cell_OV THEN

			PMS.SysBatProtect.Field.BSA_Fault_Cell_OV  := TRUE;

		ELSIF SubBMS_Calculator.BSA[LoopCount].Rack_AlarmState.Field.warning.BSA_Wn_Cell_OV THEN

			PMS.SysBatProtect.Field.BSA_Alarm_Cell_OV  := TRUE;

		END_IF;

		IF 	SubBMS_Calculator.BSA[LoopCount].Rack_AlarmState.Field.protect.BSA_Prtct_Cell_UV THEN

			PMS.SysBatProtect.Field.BSA_Prtct_Cell_UV  := TRUE;

		ELSIF SubBMS_Calculator.BSA[LoopCount].Rack_AlarmState.Field.fault.BSA_FLT_Cell_UV THEN

			PMS.SysBatProtect.Field.BSA_Fault_Cell_UV  := TRUE;

		ELSIF SubBMS_Calculator.BSA[LoopCount].Rack_AlarmState.Field.warning.BSA_Wn_Cell_UV THEN

			PMS.SysBatProtect.Field.BSA_Alarm_Cell_UV  := TRUE;

		END_IF;

		IF 	SubBMS_Calculator.BSA[LoopCount].Rack_AlarmState.Field.protect.BSA_Prtct_Cell_UnbalV THEN

			PMS.SysBatProtect.Field.BSA_Prtct_Cell_UnBalaV  := TRUE;

		ELSIF SubBMS_Calculator.BSA[LoopCount].Rack_AlarmState.Field.fault.BSA_FLT_Cell_UnbalV THEN

			PMS.SysBatProtect.Field.BSA_Prtct_Cell_UnBalaV  := TRUE;

		ELSIF SubBMS_Calculator.BSA[LoopCount].Rack_AlarmState.Field.warning.BSA_Wn_Cell_UnbalV THEN

			PMS.SysBatProtect.Field.BSA_Prtct_Cell_UnBalaV  := TRUE;

		END_IF;

		IF 	SubBMS_Calculator.BSA[LoopCount].Rack_AlarmState.Field.protect.BSA_Prtct_DisCharger_Cell_OT THEN

			PMS.SysBatProtect.Field.BSA_Prtct_Discharger_Cell_OT  := TRUE;

		ELSIF SubBMS_Calculator.BSA[LoopCount].Rack_AlarmState.Field.fault.BSA_FLT_DisCharger_Cell_OT THEN

			PMS.SysBatProtect.Field.BSA_Fault_Discharger_Cell_OT  := TRUE;

		ELSIF SubBMS_Calculator.BSA[LoopCount].Rack_AlarmState.Field.warning.BSA_Wn_DisCharger_Cell_OT THEN

			PMS.SysBatProtect.Field.BSA_Alarm_Discharger_Cell_OT  := TRUE;

		END_IF;

		IF 	SubBMS_Calculator.BSA[LoopCount].Rack_AlarmState.Field.protect.BSA_Prtct_Charger_Cell_OT THEN

			PMS.SysBatProtect.Field.BSA_Prtct_Charger_Cell_OT  := TRUE;

		ELSIF SubBMS_Calculator.BSA[LoopCount].Rack_AlarmState.Field.fault.BSA_FLT_Charger_Cell_OT THEN

			PMS.SysBatProtect.Field.BSA_Fault_Charger_Cell_OT  := TRUE;

		ELSIF SubBMS_Calculator.BSA[LoopCount].Rack_AlarmState.Field.warning.BSA_Wn_Charger_Cell_OT THEN

			PMS.SysBatProtect.Field.BSA_Alarm_Charger_Cell_OT  := TRUE;

		END_IF;

		IF 	SubBMS_Calculator.BSA[LoopCount].Rack_AlarmState.Field.protect.BSA_Prtct_DisCharger_Cell_UT THEN

			PMS.SysBatProtect.Field.BSA_Prtct_Discharger_Cell_UT  := TRUE;

		ELSIF SubBMS_Calculator.BSA[LoopCount].Rack_AlarmState.Field.fault.BSA_FLT_DisCharger_Cell_UT THEN

			PMS.SysBatProtect.Field.BSA_Fault_Discharger_Cell_UT  := TRUE;

		ELSIF SubBMS_Calculator.BSA[LoopCount].Rack_AlarmState.Field.warning.BSA_Wn_DisCharger_Cell_UT THEN

			PMS.SysBatProtect.Field.BSA_Alarm_Discharger_Cell_UT  := TRUE;

		END_IF;

		IF 	SubBMS_Calculator.BSA[LoopCount].Rack_AlarmState.Field.protect.BSA_Prtct_Charger_Cell_UT THEN

			PMS.SysBatProtect.Field.BSA_Prtct_Charger_Cell_UT  := TRUE;

		ELSIF SubBMS_Calculator.BSA[LoopCount].Rack_AlarmState.Field.fault.BSA_FLT_Charger_Cell_UT THEN

			PMS.SysBatProtect.Field.BSA_Fault_Charger_Cell_UT  := TRUE;

		ELSIF SubBMS_Calculator.BSA[LoopCount].Rack_AlarmState.Field.warning.BSA_Wn_Charger_Cell_UT THEN

			PMS.SysBatProtect.Field.BSA_Alarm_Charger_Cell_UT  := TRUE;

		END_IF;

		IF 	SubBMS_Calculator.BSA[LoopCount].Rack_AlarmState.Field.protect.BSA_Prtct_Cell_UnbalT THEN

			PMS.SysBatProtect.Field.BSA_Alarm_Cell_UnBalaT  := TRUE;

		ELSIF SubBMS_Calculator.BSA[LoopCount].Rack_AlarmState.Field.fault.BSA_FLT_Cell_UnbalT THEN

			PMS.SysBatProtect.Field.BSA_Alarm_Cell_UnBalaT  := TRUE;

		ELSIF SubBMS_Calculator.BSA[LoopCount].Rack_AlarmState.Field.warning.BSA_Wn_Cell_UnbalT THEN

			PMS.SysBatProtect.Field.BSA_Alarm_Cell_UnBalaT  := TRUE;

		END_IF;

		IF 	SubBMS_Calculator.BSA[LoopCount].Rack_AlarmState.Field.protect.BSA_Prtct_Rly_Err THEN

			PMS.SysBatProtect.Field.BSA_Prtct_RelayWelding  := TRUE;

		END_IF;
		IF 	SubBMS_Calculator.BSA[LoopCount].Rack_AlarmState.Field.protect.BSA_Prtct_IN_COM_Err  THEN

			PMS.SysBatProtect.Field.BSA_Prtct_InternalCOM   := TRUE;

		END_IF;

		IF 	SubBMS_Calculator.BSA[LoopCount].Rack_AlarmState.Field.protect.BSA_Prtct_EX_COM_Err THEN

			PMS.SysBatProtect.Field.BSA_Prtct_ExternalCOM  := TRUE;

		END_IF;

		IF 	SubBMS_Calculator.BSA[LoopCount].Rack_AlarmState.Field.protect.BSA_Prtct_Water_Leak_Err THEN

			PMS.SysBatProtect.Field.BSA_Prtct_WaterLeak  := TRUE;

		END_IF;

		IF 	SubBMS_Calculator.BSA[LoopCount].Rack_AlarmState.Field.protect.BSA_Prtct_SOC_OV THEN

			PMS.SysBatProtect.Field.BSA_Alarm_SOC_OV  := TRUE;

		END_IF;

	END_FOR;

END_ACTION

ACTION PMS_SysBatDIO:

//	PMS.SysBatDIO.Field.BSA_Prelay_DO_Status
//	PMS.SysBatDIO.Field.BSA_Nrelay_DO_Status
//	PMS.SysBatDIO.Field.BSA_ProRelay_DO_Status
//	PMS.SysBatDIO.Field.BSA_PowerLamp_DO_Status
//	PMS.SysBatDIO.Field.BSA_DO_Spare06
//	PMS.SysBatDIO.Field.BSA_DO_Spare07
//	PMS.SysBatDIO.Field.BSA_DO_Spare08
//	PMS.SysBatDIO.Field.BSA_DO_Spare09
//	PMS.SysBatDIO.Field.BSA_DO_Spare10
//	PMS.SysBatDIO.Field.BSA_DO_Spare11
//	PMS.SysBatDIO.Field.BSA_DO_Spare12
//	PMS.SysBatDIO.Field.BSA_PRelayAUX_DI_Status
//	PMS.SysBatDIO.Field.BSA_NRelayAUX_DI_Status
//	PMS.SysBatDIO.Field.BSA_EMGSwitch_DI_Status
//	PMS.SysBatDIO.Field.BSA_CoolingSystem_DI_Status
//	PMS.SysBatDIO.Field.BSA_MDS_DI_Status
//	PMS.SysBatDIO.Field.BSA_DI_Spare06
//	PMS.SysBatDIO.Field.BSA_DI_Spare07
//	PMS.SysBatDIO.Field.BSA_DI_Spare08
//	PMS.SysBatDIO.Field.BSA_DI_Spare09
//	PMS.SysBatDIO.Field.BSA_DI_Spare10
//	PMS.SysBatDIO.Field.BSA_DI_Spare11
//	PMS.SysBatDIO.Field.BSA_DI_Spare12

	PMS.SysBatDIO.Field.BSA_SOH := 0;

	FOR LoopCount := 0 TO RACK_MAXNUM_MINUS_1 DO
		PMS.SysBatDIO.Field.BSA_SOH := PMS.SysBatDIO.Field.BSA_SOH + SubBMS_Calculator.BSA[LoopCount].Rack_Calc.Field.BRA_SOH;
	END_FOR;
	IF  HMI.DeviceLoading.SetRackNum <> 0 THEN
		PMS.SysBatDIO.Field.BSA_SOH  := PMS.SysBatDIO.Field.BSA_SOH / HMI.DeviceLoading.SetRackNum ;
	END_IF;

END_ACTION

ACTION PMS_BRACal:

	PMS.BRACal.Field.BRA_Rack_Num					:=	UDINT_TO_UINT(HMI.RackIndex)+1;

	PMS.BRACal.Field.BRA_Volt_Total					:=	SubBMS_Calculator.BSA[HMI.RackIndex].Rack_Calc.Field.BRA_Volt_Total ;
	PMS.BRACal.Field.BRA_Curr_Total					:=	SubBMS_Calculator.BSA[HMI.RackIndex].Rack_Calc.Field.BRA_Curr_Total ;
	PMS.BRACal.Field.BRA_SOC						:= 	SubBMS_Calculator.BSA[HMI.RackIndex].Rack_Calc.Field.BRA_SOC ;

END_ACTION
ACTION PMS_BRAPWR_A:

	PMS.BRAPWR_A.Field.BRA_Rack_Num					:=	UDINT_TO_UINT(HMI.RackIndex)+1;
	PMS.BRAPWR_A.Field.BRA_SOH						:=	SubBMS_Calculator.BSA[HMI.RackIndex].Rack_Calc.Field.BRA_SOH ;
	PMS.BRAPWR_A.Field.BRA_CONT_CHA_PWR_Limit		:=	SubBMS_Calculator.BSA[HMI.RackIndex].Rack_PWRCalc.Field.BSA_CHAPWCont ;
	PMS.BRAPWR_A.Field.BRA_Peak_CHA_PWR_Limit		:=	SubBMS_Calculator.BSA[HMI.RackIndex].Rack_PWRCalc.Field.BSA_CHAPWPeak ;

END_ACTION
ACTION PMS_BRAPWR_B:

	PMS.BRAPWR_B.Field.BRA_Rack_Num					:=	UDINT_TO_UINT(HMI.RackIndex)+1;
	PMS.BRAPWR_B.Field.BRA_CONT_DisCHA_PWR_Limit	:=	SubBMS_Calculator.BSA[HMI.RackIndex].Rack_PWRCalc.Field.BSA_DisCHAPWCont ;
	PMS.BRAPWR_B.Field.BRA_Peak_DisCHA_PWR_Limit	:=	SubBMS_Calculator.BSA[HMI.RackIndex].Rack_PWRCalc.Field.BSA_DisCHAPWPeak ;

END_ACTION
ACTION PMS_BRACellV:

	PMS.BRACellV.Field.BRA_Rack_Num					:=	UDINT_TO_UINT(HMI.RackIndex)+1;
	PMS.BRACellV.Field.BRA_Cell_Max_Voltage			:=	SubBMS_Calculator.BSA[HMI.RackIndex].Rack_Cell_Vcalc.Field.BSA_Cell_MaxV ;
	PMS.BRACellV.Field.BRA_Cell_Min_Voltage			:=	SubBMS_Calculator.BSA[HMI.RackIndex].Rack_Cell_Vcalc.Field.BSA_Cell_MinV ;
	PMS.BRACellV.Field.BRA_Cell_AGV_Voltage			:=	SubBMS_Calculator.BSA[HMI.RackIndex].Rack_Cell_Vcalc.Field.BSA_Cell_AVGV ;

END_ACTION
ACTION PMS_BRACellT:

	PMS.BRACellT.Field.BRA_Rack_Num					:=	UDINT_TO_UINT(HMI.RackIndex)+1;
	PMS.BRACellT.Field.BRA_Cell_Max_Temperature		:=	SubBMS_Calculator.BSA[HMI.RackIndex].Rack_Cell_Tcalc.Field.BSA_Cell_MaxT ;
	PMS.BRACellT.Field.BRA_Cell_Min_Temperature		:=	SubBMS_Calculator.BSA[HMI.RackIndex].Rack_Cell_Tcalc.Field.BSA_Cell_MinT ;
	PMS.BRACellT.Field.BRA_Cell_AGV_Temperature		:=	SubBMS_Calculator.BSA[HMI.RackIndex].Rack_Cell_Tcalc.Field.BSA_Cell_AVGT ;

END_ACTION
ACTION PMS_BRACellDiv:

	PMS.BRACellDiv.Field.BRA_Rack_Num				:=	UDINT_TO_UINT(HMI.RackIndex)+1;
	PMS.BRACellDiv.Field.BRA_Cell_DIV_Voltage		:=	SubBMS_Calculator.BSA[HMI.RackIndex].Rack_Cell_Tcalc.Field.BSA_Cell_DeviT ;
	PMS.BRACellDiv.Field.BRA_Cell_DIV_Temperature	:=	SubBMS_Calculator.BSA[HMI.RackIndex].Rack_Cell_Vcalc.Field.BSA_Cell_DeviV ;

END_ACTION
ACTION PMS_BRA_VTPos:

	PMS.BRA_VTPos.Field.BRA_Rack_Num					:=	UDINT_TO_UINT(HMI.RackIndex)+1;
	PMS.BRA_VTPos.Field.BRA_Max_Cell_V_Location	:=	UINT_TO_USINT(SubBMS_Calculator.BSA[HMI.RackIndex].Rack_Cell_Pcalc.Field.BSA_Cell_MaxV_Location) ;
	PMS.BRA_VTPos.Field.BRA_Min_Cell_V_Location	:=	UINT_TO_USINT(SubBMS_Calculator.BSA[HMI.RackIndex].Rack_Cell_Pcalc.Field.BSA_Cell_MinV_Location) ;
	PMS.BRA_VTPos.Field.BRA_Max_Cell_T_Location	:=	UINT_TO_USINT(SubBMS_Calculator.BSA[HMI.RackIndex].Rack_Cell_Pcalc.Field.BSA_Cell_MaxT_Location) ;
	PMS.BRA_VTPos.Field.BRA_Min_Cell_T_Location	:=	UINT_TO_USINT(SubBMS_Calculator.BSA[HMI.RackIndex].Rack_Cell_Pcalc.Field.BSA_Cell_MinT_Location) ;

END_ACTION
ACTION PMS_BAR_Alarm:

	PMS.BAR_Alarm.Field.BRA_Rack_Num					:=	UDINT_TO_UINT(HMI.RackIndex)+1;
	//	PMS.BAR_Alarm.Field.BRA_Alarm_OC				:=	SubBMS_Calculator.BSA[HMI.RackIndex].Rack_AlarmState.Field.warning.
	PMS.BAR_Alarm.Field.BRA_Alarm_SOC_OV				:=	SubBMS_Calculator.BSA[HMI.RackIndex].Rack_AlarmState.Field.warning.BSA_Wn_SOC_OV;
	PMS.BAR_Alarm.Field.BRA_Fault_SOC_UN				:=	SubBMS_Calculator.BSA[HMI.RackIndex].Rack_AlarmState.Field.warning.BSA_Wn_SOC_Un;
	PMS.BAR_Alarm.Field.BRA_Alarm_OV					:=	SubBMS_Calculator.BSA[HMI.RackIndex].Rack_AlarmState.Field.warning.BSA_Wn_OV;
	PMS.BAR_Alarm.Field.BRA_Alarm_UV					:=	SubBMS_Calculator.BSA[HMI.RackIndex].Rack_AlarmState.Field.warning.BSA_Wn_UV;
	PMS.BAR_Alarm.Field.BRA_Alarm_Cell_OV				:=	SubBMS_Calculator.BSA[HMI.RackIndex].Rack_AlarmState.Field.warning.BSA_Wn_Cell_OV;
	PMS.BAR_Alarm.Field.BRA_Alarm_Cell_UV				:=	SubBMS_Calculator.BSA[HMI.RackIndex].Rack_AlarmState.Field.warning.BSA_Wn_Cell_UV;
	PMS.BAR_Alarm.Field.BRA_Alarm_Cell_UnBalaV			:=	SubBMS_Calculator.BSA[HMI.RackIndex].Rack_AlarmState.Field.warning.BSA_Wn_Cell_UnbalV;
	PMS.BAR_Alarm.Field.BRA_Alarm_Discharger_Cell_OT	:=	SubBMS_Calculator.BSA[HMI.RackIndex].Rack_AlarmState.Field.warning.BSA_Wn_DisCharger_Cell_OT;
	PMS.BAR_Alarm.Field.BRA_Alarm_Charger_Cell_OT		:=	SubBMS_Calculator.BSA[HMI.RackIndex].Rack_AlarmState.Field.warning.BSA_Wn_Charger_Cell_OT;
	PMS.BAR_Alarm.Field.BRA_Alarm_Charger_Cell_UT		:=	SubBMS_Calculator.BSA[HMI.RackIndex].Rack_AlarmState.Field.warning.BSA_Wn_Charger_Cell_UT;
	PMS.BAR_Alarm.Field.BRA_Alarm_Cell_UnBalaT			:=	SubBMS_Calculator.BSA[HMI.RackIndex].Rack_AlarmState.Field.warning.BSA_Wn_Cell_UnbalT;
	//	PMS.BAR_Alarm.Field.BRA_Alarm_Continuously_OP	:=	SubBMS_Calculator.BSA[HMI.RackIndex].Rack_AlarmState.Field.warning.
	//	PMS.BAR_Alarm.Field.BRA_Alarm_Peak_OP			:=	SubBMS_Calculator.BSA[HMI.RackIndex].Rack_AlarmState.Field.warning.
	//	PMS.BAR_Alarm.Field.BRA_Fault_OC				:=	SubBMS_Calculator.BSA[HMI.RackIndex].Rack_AlarmState.Field.fault.
	PMS.BAR_Alarm.Field.BRA_Fault_SOC_OV				:=	SubBMS_Calculator.BSA[HMI.RackIndex].Rack_AlarmState.Field.fault.BSA_FLT_SOC_OV;
	PMS.BAR_Alarm.Field.BRA_Fault_SOC_UN				:=	SubBMS_Calculator.BSA[HMI.RackIndex].Rack_AlarmState.Field.fault.BSA_FLT_SOC_Un;
	PMS.BAR_Alarm.Field.BRA_Fault_OV					:=	SubBMS_Calculator.BSA[HMI.RackIndex].Rack_AlarmState.Field.fault.BSA_FLT_OV;
	PMS.BAR_Alarm.Field.BRA_Fault_UV					:=	SubBMS_Calculator.BSA[HMI.RackIndex].Rack_AlarmState.Field.fault.BSA_FLT_UV;
	PMS.BAR_Alarm.Field.BRA_Fault_Cell_OV				:=	SubBMS_Calculator.BSA[HMI.RackIndex].Rack_AlarmState.Field.fault.BSA_FLT_Cell_OV;
	PMS.BAR_Alarm.Field.BRA_Fault_Cell_UV				:=	SubBMS_Calculator.BSA[HMI.RackIndex].Rack_AlarmState.Field.fault.BSA_FLT_Cell_UV;
	PMS.BAR_Alarm.Field.BRA_Fault_Cell_UnBalaV			:=	SubBMS_Calculator.BSA[HMI.RackIndex].Rack_AlarmState.Field.fault.BSA_FLT_Cell_UnbalV;
	PMS.BAR_Alarm.Field.BRA_Fault_Discharger_Cell_OT	:=	SubBMS_Calculator.BSA[HMI.RackIndex].Rack_AlarmState.Field.fault.BSA_FLT_DisCharger_Cell_OT;
	PMS.BAR_Alarm.Field.BRA_Fault_Charger_Cell_OT		:=	SubBMS_Calculator.BSA[HMI.RackIndex].Rack_AlarmState.Field.fault.BSA_FLT_Charger_Cell_OT;
	PMS.BAR_Alarm.Field.BRA_Fault_Charger_Cell_UT		:=	SubBMS_Calculator.BSA[HMI.RackIndex].Rack_AlarmState.Field.fault.BSA_FLT_Charger_Cell_UT;
	PMS.BAR_Alarm.Field.BRA_Fault_Cell_UnBalaT			:=	SubBMS_Calculator.BSA[HMI.RackIndex].Rack_AlarmState.Field.fault.BSA_FLT_Cell_UnbalT;
	//	PMS.BAR_Alarm.Field.BRA_Fault_Continuously_OP	:=	SubBMS_Calculator.BSA[HMI.RackIndex].Rack_AlarmState.Field.fault.
	//	PMS.BAR_Alarm.Field.BRA_Fault_Peak_OP			:=	SubBMS_Calculator.BSA[HMI.RackIndex].Rack_AlarmState.Field.fault.

END_ACTION
ACTION PMS_BAR_Protect:

	PMS.BAR_Protect.Field.BRA_Rack_Num					:=	UDINT_TO_UINT(HMI.RackIndex)+1;
	//	PMS.BAR_Protect.Field.BRA_Prtct_OC					:=	SubBMS_Calculator.BSA[HMI.RackIndex].Rack_AlarmState.Field.warning.
	PMS.BAR_Protect.Field.BRA_Prtct_SOC_OV				:=	SubBMS_Calculator.BSA[HMI.RackIndex].Rack_AlarmState.Field.protect.BSA_Prtct_SOC_OV;
	PMS.BAR_Protect.Field.BRA_Prtct_SOC_UN				:=	SubBMS_Calculator.BSA[HMI.RackIndex].Rack_AlarmState.Field.protect.BSA_Prtct_SOC_Un;
	PMS.BAR_Protect.Field.BRA_Prtct_OV					:=	SubBMS_Calculator.BSA[HMI.RackIndex].Rack_AlarmState.Field.protect.BSA_Prtct_OV;
	PMS.BAR_Protect.Field.BRA_Prtct_UV					:=	SubBMS_Calculator.BSA[HMI.RackIndex].Rack_AlarmState.Field.protect.BSA_Prtct_UV;
	PMS.BAR_Protect.Field.BRA_Prtct_Cell_OV				:=	SubBMS_Calculator.BSA[HMI.RackIndex].Rack_AlarmState.Field.protect.BSA_Prtct_Cell_OV;
	PMS.BAR_Protect.Field.BRA_Prtct_Cell_UV				:=	SubBMS_Calculator.BSA[HMI.RackIndex].Rack_AlarmState.Field.protect.BSA_Prtct_Cell_UV;
	PMS.BAR_Protect.Field.BRA_Prtct_Cell_UnBalaV		:=	SubBMS_Calculator.BSA[HMI.RackIndex].Rack_AlarmState.Field.protect.BSA_Prtct_Cell_UnbalV;
	PMS.BAR_Protect.Field.BRA_Prtct_Discharger_Cell_OT	:=	SubBMS_Calculator.BSA[HMI.RackIndex].Rack_AlarmState.Field.protect.BSA_Prtct_DisCharger_Cell_OT;
	PMS.BAR_Protect.Field.BRA_Prtct_Charger_Cell_OT		:=	SubBMS_Calculator.BSA[HMI.RackIndex].Rack_AlarmState.Field.protect.BSA_Prtct_Charger_Cell_OT;
	PMS.BAR_Protect.Field.BRA_Prtct_Charger_Cell_UT		:=	SubBMS_Calculator.BSA[HMI.RackIndex].Rack_AlarmState.Field.protect.BSA_Prtct_Charger_Cell_UT;
	PMS.BAR_Protect.Field.BRA_Prtct_Cell_UnBalaT		:=	SubBMS_Calculator.BSA[HMI.RackIndex].Rack_AlarmState.Field.protect.BSA_Prtct_Cell_UnbalT;
	//	PMS.BAR_Protect.Field.BRA_Prtct_Continuously_OP		:=	SubBMS_Calculator.BSA[HMI.RackIndex].Rack_AlarmState.Field.protect.
	//	PMS.BAR_Protect.Field.BRA_Prtct_Peak_OP				:=	SubBMS_Calculator.BSA[HMI.RackIndex].Rack_AlarmState.Field.protect.
	PMS.BAR_Protect.Field.BRA_Prtct_InternalCOM			:=	SubBMS_Calculator.BSA[HMI.RackIndex].Rack_AlarmState.Field.protect.BSA_Prtct_IN_COM_Err;
	PMS.BAR_Protect.Field.BRA_Prtct_ExternalCOM			:=	SubBMS_Calculator.BSA[HMI.RackIndex].Rack_AlarmState.Field.protect.BSA_Prtct_EX_COM_Err;
	PMS.BAR_Protect.Field.BRA_Prtct_RelayWelding		:=	SubBMS_Calculator.BSA[HMI.RackIndex].Rack_AlarmState.Field.protect.BSA_Prtct_Rly_Err;
	PMS.BAR_Protect.Field.BRA_Prtct_WaterLeak			:=	SubBMS_Calculator.BSA[HMI.RackIndex].Rack_AlarmState.Field.protect.BSA_Prtct_Water_Leak_Err;
	//	PMS.BAR_Protect.Field.BRA_Prtct_InsulationReg		:=	SubBMS_Calculator.BSA[HMI.RackIndex].Rack_AlarmState.Field.protect.BSA_Prtct_Cell_OV;
	//	PMS.BAR_Protect.Field.BRA_Prtct_MDSFuse				:=	SubBMS_Calculator.BSA[HMI.RackIndex].Rack_AlarmState.Field.protect.BSA_Prtct_Cell_UV;
	//	PMS.BAR_Protect.Field.BRA_Prtct_CoolingSystem		:=	SubBMS_Calculator.BSA[HMI.RackIndex].Rack_AlarmState.Field.protect.BSA_Prtct_Cell_UnbalV;

END_ACTION
ACTION PMS_BAR_DIO:

	PMS.BAR_DIO.Field.BRA_Rack_Num						:=	UDINT_TO_UINT(HMI.RackIndex)+1;
	//	PMS.BAR_DIO.Field.BRA_CONT_DisCHA_PWR_Limit			:=	SubBMS_Calculator.BSA[HMI.RackIndex].Rack_Calc.Field.BRA_Volt_Total
	//	PMS.BAR_DIO.Field.BRA_Peak_DisCHA_PWR_Limit			:=	SubBMS_Calculator.BSA[HMI.RackIndex].Rack_Calc.Field.BRA_Curr_Total
	//	PMS.BAR_DIO.Field.BRA_Prelay_DO_Status 				:=	SubBMS_Calculator.BSA[HMI.RackIndex].Rack_Calc.Field.BRA_Volt_Total
	//	PMS.BAR_DIO.Field.BRA_Nrelay_DO_Status 				:=	SubBMS_Calculator.BSA[HMI.RackIndex].Rack_Calc.Field.BRA_Volt_Total
	//	PMS.BAR_DIO.Field.BRA_ProRelay_DO_Status 			:=	SubBMS_Calculator.BSA[HMI.RackIndex].Rack_Calc.Field.BRA_Volt_Total
	//	PMS.BAR_DIO.Field.BRA_PowerLamp_DO_Status 			:=	SubBMS_Calculator.BSA[HMI.RackIndex].Rack_Calc.Field.BRA_Volt_Total
	//	PMS.BAR_DIO.Field.BRA_Buzzer_DO_Status				:=	SubBMS_Calculator.BSA[HMI.RackIndex].Rack_Calc.Field.BRA_Volt_Total
	//	PMS.BAR_DIO.Field.BRA_PRelayAUX_DI_Status			:=	SubBMS_Calculator.BSA[HMI.RackIndex].Rack_Calc.Field.BRA_Volt_Total
	//	PMS.BAR_DIO.Field.BRA_NRelayAUX_DI_Status 			:=	SubBMS_Calculator.BSA[HMI.RackIndex].Rack_Calc.Field.BRA_Volt_Total
	//	PMS.BAR_DIO.Field.BRA_EMGSwitch_DI_Status 			:=	SubBMS_Calculator.BSA[HMI.RackIndex].Rack_Calc.Field.BRA_Volt_Total
	//	PMS.BAR_DIO.Field.BRA_MDS_DI_Status					:=	SubBMS_Calculator.BSA[HMI.RackIndex].Rack_Calc.Field.BRA_Volt_Total
	PMS.BAR_DIO.Field.BRA_Waterleak_Dete_MD1			:=	SubBMS_Calculator.BSA[HMI.RackIndex].Modul1_Info.Field.OPS_Waterleak_Err ;
	PMS.BAR_DIO.Field.BRA_Waterleak_Dete_MD2			:=	SubBMS_Calculator.BSA[HMI.RackIndex].Modul2_Info.Field.OPS_Waterleak_Err ;
	PMS.BAR_DIO.Field.BRA_Waterleak_Dete_MD3			:=	SubBMS_Calculator.BSA[HMI.RackIndex].Modul3_Info.Field.OPS_Waterleak_Err ;
	PMS.BAR_DIO.Field.BRA_Waterleak_Dete_MD4			:=	SubBMS_Calculator.BSA[HMI.RackIndex].Modul4_Info.Field.OPS_Waterleak_Err ;
	PMS.BAR_DIO.Field.BRA_Waterleak_Dete_MD5			:=	SubBMS_Calculator.BSA[HMI.RackIndex].Modul5_Info.Field.OPS_Waterleak_Err ;
	PMS.BAR_DIO.Field.BRA_Waterleak_Dete_MD6			:=	SubBMS_Calculator.BSA[HMI.RackIndex].Modul6_Info.Field.OPS_Waterleak_Err ;
	PMS.BAR_DIO.Field.BRA_Waterleak_Dete_MD7			:=	SubBMS_Calculator.BSA[HMI.RackIndex].Modul7_Info.Field.OPS_Waterleak_Err ;

END_ACTION
```

#### System_HMI.st
```iecst
ACTION System_RackState:
	FOR LoopCount := 0 TO RACK_MAXNUM_MINUS_1 DO

		CASE SubBMS_Calculator.BSA[LoopCount].Rack_State.Field.BSA_Divice_Status OF
			0:  HMI.SystemRackInfo.RACK_State[LoopCount] := 'NONE';
			1:  HMI.SystemRackInfo.RACK_State[LoopCount] := 'IDEL';
			2:  HMI.SystemRackInfo.RACK_State[LoopCount] := 'STANDBY';
			3:  HMI.SystemRackInfo.RACK_State[LoopCount] := 'READY';
			4:  HMI.SystemRackInfo.RACK_State[LoopCount] := 'RUN';
			5:  HMI.SystemRackInfo.RACK_State[LoopCount] := 'PROTECT';
			6:  HMI.SystemRackInfo.RACK_State[LoopCount] := 'STOP';
		END_CASE;
	END_FOR;
END_ACTION

ACTION System_RackVolt:
	FOR LoopCount := 0 TO RACK_MAXNUM_MINUS_1 DO
			HMI.SystemRackInfo.RACK_BRA_Volt_Total[LoopCount] := REAL_TO_STRING((SubBMS_Calculator.BSA[LoopCount].Rack_Calc.Field.BRA_Volt_Total));
	END_FOR;
END_ACTION

ACTION System_RackCurr:
	FOR LoopCount := 0 TO RACK_MAXNUM_MINUS_1 DO

			HMI.SystemRackInfo.RACK_BRA_Curr_Total[LoopCount] := REAL_TO_STRING((SubBMS_Calculator.BSA[LoopCount].Rack_Calc.Field.BRA_Curr_Total));
	END_FOR;
END_ACTION

ACTION System_RackTotal:
	FOR LoopCount := 0 TO RACK_MAXNUM_MINUS_1 DO

		IF HMI.RackEnable[LoopCount] THEN
			HMI.SystemRackInfo.RACK_BRA_Total[LoopCount] := CONCAT(HMI.SystemRackInfo.RACK_BRA_Volt_Total[LoopCount],CONCAT('(V), ',CONCAT(HMI.SystemRackInfo.RACK_BRA_Curr_Total[LoopCount],'(A)')));
		ELSE
			HMI.SystemRackInfo.RACK_BRA_Total[LoopCount] := 'Not Used';
		END_IF;
	END_FOR;
END_ACTION
```

### Program Logical/Source/PMS_MODBUS/ModbusPMS (IEC)

#### Main.st
```iecst
PROGRAM _INIT

	ModbusCtrl.Init_Parameter.ModbusStation					:= 'IF2.MODBUSSLAVE_1' ;
	ModbusCtrl.Init_Parameter.register_StartAddress			:= 0 ;
	ModbusCtrl.Init_Parameter.FunctionNum					:= mbMFC_READ_INPUT_REGISTERS ;
	ModbusCtrl.Init_Parameter.RegisterNum					:= 72;

	fub_status			:= 0;							(* status of function blocks *)
	mb_exception		:= 0;							(* modbus exception *)

END_PROGRAM

PROGRAM _CYCLIC

	(* WORKING STATE MACHINE *)	// 16 BIT << CAN DATA 64 BIT
	memcpy(ADR(ModbusCtrl.Data.Register[0]),ADR(PMS.SysBatProduct.Value),SIZEOF(PMS.SysBatProduct.Value));
	memcpy(ADR(ModbusCtrl.Data.Register[4]),ADR(PMS.SysBatCal.Value),SIZEOF(PMS.SysBatCal.Value));
	memcpy(ADR(ModbusCtrl.Data.Register[8]),ADR(PMS.SysBatPWR.Value),SIZEOF(PMS.SysBatPWR.Value));
	memcpy(ADR(ModbusCtrl.Data.Register[12]),ADR(PMS.SysCellVolt.Value),SIZEOF(PMS.SysCellVolt.Value));
	memcpy(ADR(ModbusCtrl.Data.Register[16]),ADR(PMS.SysCellTemps.Value),SIZEOF(PMS.SysCellTemps.Value));
	memcpy(ADR(ModbusCtrl.Data.Register[20]),ADR(PMS.SysCellV_TPos.Value),SIZEOF(PMS.SysCellV_TPos.Value));
	memcpy(ADR(ModbusCtrl.Data.Register[24]),ADR(PMS.SysBatProtect.Value),SIZEOF(PMS.SysBatProtect.Value));
	memcpy(ADR(ModbusCtrl.Data.Register[28]),ADR(PMS.SysBatDIO.Value),SIZEOF(PMS.SysBatDIO.Value));
	memcpy(ADR(ModbusCtrl.Data.Register[32]),ADR(PMS.BRACal.Value),SIZEOF(PMS.BRACal.Value));
	memcpy(ADR(ModbusCtrl.Data.Register[36]),ADR(PMS.BRAPWR_A.Value),SIZEOF(PMS.BRAPWR_A.Value));
	memcpy(ADR(ModbusCtrl.Data.Register[40]),ADR(PMS.BRAPWR_B.Value),SIZEOF(PMS.BRAPWR_B.Value));
	memcpy(ADR(ModbusCtrl.Data.Register[44]),ADR(PMS.BRACellV.Value),SIZEOF(PMS.BRACellV.Value));
	memcpy(ADR(ModbusCtrl.Data.Register[48]),ADR(PMS.BRACellT.Value),SIZEOF(PMS.BRACellT.Value));
	memcpy(ADR(ModbusCtrl.Data.Register[52]),ADR(PMS.BRACellDiv.Value),SIZEOF(PMS.BRACellDiv.Value));
	memcpy(ADR(ModbusCtrl.Data.Register[56]),ADR(PMS.BRA_VTPos.Value),SIZEOF(PMS.BRA_VTPos.Value));
	memcpy(ADR(ModbusCtrl.Data.Register[60]),ADR(PMS.BAR_Alarm.Value),SIZEOF(PMS.BAR_Alarm.Value));
	memcpy(ADR(ModbusCtrl.Data.Register[64]),ADR(PMS.BAR_Protect.Value),SIZEOF(PMS.BAR_Protect.Value));
	memcpy(ADR(ModbusCtrl.Data.Register[68]),ADR(PMS.BAR_DIO.Value),SIZEOF(PMS.BAR_DIO.Value));

	CASE (ModbusCtrl.Init_Parameter.FunctionNum) OF
		mbMFC_READ_INPUT_REGISTERS:

			ModbusCtrl.Write_Multiple_Registers(enable := TRUE,
				startAddress := 30001,
			nrOfItems := ModbusCtrl.Init_Parameter.RegisterNum,
			station := ModbusCtrl.Init_Parameter.ModbusStation,
			data := ModbusCtrl.Data.Register);

			IF (ModbusCtrl.Read_Holding_Registers.status <> ERR_FUB_BUSY) THEN
				fub_status 			:= ModbusCtrl.Write_Multiple_Registers.status;

				check_status 		:= TRUE;			(* flag to check status *)
				instruction_ready 	:= TRUE;			(* flag marks instruction "ready" *)
			ELSE

			END_IF

		mbMFC_READ_HOLDING_REGISTERS: 	// Modbus Function 03

			ModbusCtrl.Read_Holding_Registers(enable := TRUE,
				startAddress := 40001,
				nrOfItems := 1,
			station := ModbusCtrl.Init_Parameter.ModbusStation,
			data := ModbusCtrl.Data.Register);

//			Modbus.BSA_WakeUp_CMD 	:= ModbusCtrl.Data.Register[0].0;
//			Modbus.BSA_POWER_CMD	:= ModbusCtrl.Data.Register[0].1;
//			Modbus.BSA_FaultReset	:= ModbusCtrl.Data.Register[0].8;

			IF (ModbusCtrl.Read_Holding_Registers.status <> ERR_FUB_BUSY) THEN
				fub_status 			:= ModbusCtrl.Write_Multiple_Registers.status;

				check_status 		:= TRUE;			(* flag to check status *)
				instruction_ready 	:= TRUE;			(* flag marks instruction "ready" *)
			ELSE

			END_IF

	END_CASE

	(* ERROR HANDLING *)
	IF (check_status) THEN

		CASE fub_status OF

			ERR_OK:

				gSignalCheck.TCP_Check := TRUE;

			ELSE
				(* other error handling *)

		END_CASE;

		(* stop checking *)
		check_status := FALSE;
	END_IF

	//
	//	(* STATE MACHINE CONTROL *)
	//	IF (instruction_ready AND fub_status = ERR_OK) THEN
	//
	//		CASE (instruction) OF
	//
	//			mbMFC_READ_HOLDING_REGISTERS:
	//				instruction 		:= mbMFC_READ_COILS;
	//				instruction_ready 	:= FALSE;
	//
	//			mbMFC_READ_COILS:
	//				instruction 		:= mbMFC_READ_HOLDING_REGISTERS;
	//				instruction_ready 	:= FALSE;
	//
	//		END_CASE
	//
	//	END_IF

END_PROGRAM
```

### Program Logical/Source/HMI/HMI_DataParsing (IEC)

#### Main.st - Init, cyclic, exit code
```iecst
PROGRAM _INIT
	HMI;

	Timestamp.DTGetTime_0.enable := TRUE;

	HMI_AlarmName[0] := 'Sys Over Current';
	HMI_AlarmName[1] := 'Sys Over SOC';
	HMI_AlarmName[2] := 'Sys Under SOC';
	HMI_AlarmName[3] := 'Sys Over Voltage';
	HMI_AlarmName[4] := 'Sys Under Voltag';
	HMI_AlarmName[5] := 'Cell Over Voltage';
	HMI_AlarmName[6] := 'Cell Under Voltag';
	HMI_AlarmName[7] := 'Cell UnBalance Voltage';
	HMI_AlarmName[8] := 'Cell DisCHA Over Temperature';
	HMI_AlarmName[9] := 'Cell CHA Over Temperature';
	HMI_AlarmName[10] := 'Cell DisCHA Under Temperature';
	HMI_AlarmName[11] := 'Cell CHA Under Temperature';
	HMI_AlarmName[12] := 'Cell UnBalance Temperature';

	HMI_AlarmName[13] := 'Relay Welding Error';
	HMI_AlarmName[14] := 'Internal COM Error';
	HMI_AlarmName[15] := 'External COM Error';
	HMI_AlarmName[16] := 'Current Transformer COM Error';
	HMI_AlarmName[17] := 'Water Leak Error';
	HMI_AlarmName[18] := 'Emergency Switch Error';

	FOR LoopNum := 0 TO 12 DO

		HMI_Alarm.Warning[LoopNum].Name 	:=	HMI_AlarmName[LoopNum];
		HMI_Alarm.Fault[LoopNum].Name 		:=	HMI_AlarmName[LoopNum];
		HMI_Alarm.Protect[LoopNum].Name 	:=	HMI_AlarmName[LoopNum];

	END_FOR;

	FOR LoopNum := 13 TO 18 DO

		HMI_Alarm.Protect[LoopNum].Name 	:=	HMI_AlarmName[LoopNum];

	END_FOR;
END_PROGRAM

PROGRAM _CYCLIC

	ActTimeSplit;
	ActSystem_Warning;
	ActSystem_Fault;
	ActSystem_Protect;
	ActLOGIN;
	ActSystem_AlarmTab;
	ActDeviceReset;

	CASE HMI.Step OF
		vkINITIAL:
			HMI.Step := vkBOOTING;
		vkBOOTING:
		vkSYSTEM:
			memcpy(ADR(System_HMI),ADR(PMS),SIZEOF(PMS));
			HMI.RackIndex := vkRACKNUM1;
			AtSystemUI;
		vkRACK1:
			memcpy(ADR(Rack_HMI),ADR(SubBMS.Rack1.BSA),SIZEOF(Rack_HMI));
			HMI.RackIndex := vkRACKNUM1;
			AtRackUI;
		vkRACK2:
			memcpy(ADR(Rack_HMI),ADR(SubBMS.Rack2.BSA),SIZEOF(Rack_HMI));
			HMI.RackIndex := vkRACKNUM2;
			AtRackUI;
		vkRACK3:
			memcpy(ADR(Rack_HMI),ADR(SubBMS.Rack3.BSA),SIZEOF(Rack_HMI));
			HMI.RackIndex := vkRACKNUM3;
			AtRackUI;
		vkRACK4:
			memcpy(ADR(Rack_HMI),ADR(SubBMS.Rack4.BSA),SIZEOF(Rack_HMI));
			HMI.RackIndex := vkRACKNUM4;
			AtRackUI;
		vkALARMHISTORY:
			memcpy(ADR(System_HMI),ADR(PMS),SIZEOF(PMS));
			AtSystemUI;
		vkADMINISTRATOR:
			memcpy(ADR(System_HMI),ADR(PMS),SIZEOF(PMS));
			AtSystemUI;

	END_CASE;
END_PROGRAM

PROGRAM _EXIT
	(* Insert code here *)
END_PROGRAM
```

#### Variables.var - Local variables
```iecst
VAR
	strStyleLED_CAN_1 : STRING[40];
	countTime_0 : USINT;
END_VAR
(*Insert your comment here.*)
(*Insert your comment here.*)
VAR
	TON_0 : TON;
	Timestamp : TimeType;
	LoopNum : INT;
END_VAR
```

#### HMI_Rack.st
```iecst
ACTION AtRackUI :

	CASE Rack_HMI.Rack_State.Field.BSA_Divice_Status OF
		0:  HMI.BSA_Divice_Status := 'NONE';
		1:  HMI.BSA_Divice_Status := 'IDEL';
		2:  HMI.BSA_Divice_Status := 'STANDBY';
		3:  HMI.BSA_Divice_Status := 'READY';
		4:  HMI.BSA_Divice_Status := 'RUN';
		5:  HMI.BSA_Divice_Status := 'PROTECT';
		6:  HMI.BSA_Divice_Status := 'STOP';
	END_CASE;

	HMI.Gauge.BRA_Volt_Total		:= (Rack_HMI.Rack_Calc.Field.BRA_Volt_Total) ;
	HMI.Gauge.BRA_Volt_Total_A		:= REAL_TO_STRING((HMI.Gauge.BRA_Volt_Total-400)*0.675);
	HMI.Gauge.BRA_Volt_Total_B		:= CONCAT('[{"select":"#gauge3","spin":[',CONCAT(HMI.Gauge.BRA_Volt_Total_A,',0,0]}]'));

	HMI.Gauge.BRA_Curr_Total 			:= (Rack_HMI.Rack_Calc.Field.BRA_Curr_Total) ;
	HMI.Gauge.BRA_Curr_Total_A		:= REAL_TO_STRING(HMI.Gauge.BRA_Curr_Total*0.27+135);
	HMI.Gauge.BRA_Curr_Total_B		:= CONCAT('[{"select":"#gauge4","spin":[',CONCAT(HMI.Gauge.BRA_Curr_Total_A,',0,0]}]'));

	HMI.Gauge.BRA_SOC		:= (Rack_HMI.Rack_Calc.Field.BRA_SOC)  ;
	HMI.Gauge.BRA_SOC_A		:= REAL_TO_STRING(HMI.Gauge.BRA_SOC*2.7);
	HMI.Gauge.BRA_SOC_B		:= CONCAT('[{"select":"#gauge1","spin":[',CONCAT(HMI.Gauge.BRA_SOC_A,',0,0]}]'));

	HMI.Gauge.BRA_SOH		:= (Rack_HMI.Rack_Calc.Field.BRA_SOH) ;
	HMI.Gauge.BRA_SOH_A		:= REAL_TO_STRING(HMI.Gauge.BRA_SOH*2.7);
	HMI.Gauge.BRA_SOH_B		:= CONCAT('[{"select":"#gauge2","spin":[',CONCAT(HMI.Gauge.BRA_SOH_A,',0,0]}]'));

	HMI.BatteryInfo.BSA_Cell_MaxV 		:= (Rack_HMI.Rack_Cell_Vcalc.Field.BSA_Cell_MaxV);
	HMI.BatteryInfo.BSA_Cell_MinV		:= (Rack_HMI.Rack_Cell_Vcalc.Field.BSA_Cell_MinV) ;
	HMI.BatteryInfo.BSA_Cell_AVGV		:= (Rack_HMI.Rack_Cell_Vcalc.Field.BSA_Cell_AVGV)  ;
	HMI.BatteryInfo.BSA_Cell_DeviV 		:= (Rack_HMI.Rack_Cell_Vcalc.Field.BSA_Cell_DeviV)  ;

	HMI.BatteryInfo.BSA_Cell_MaxT 		:= (Rack_HMI.Rack_Cell_Tcalc.Field.BSA_Cell_MaxT)  ;
	HMI.BatteryInfo.BSA_Cell_MinT		:= (Rack_HMI.Rack_Cell_Tcalc.Field.BSA_Cell_MinT	) ;
	HMI.BatteryInfo.BSA_Cell_AVGT		:= (Rack_HMI.Rack_Cell_Tcalc.Field.BSA_Cell_AVGT)  ;
	HMI.BatteryInfo.BSA_Cell_DeviT 		:= (Rack_HMI.Rack_Cell_Tcalc.Field.BSA_Cell_DeviT) ;

	HMI.BatteryInfo.BSA_Cell_MaxV_Cell_Location		:= UINT_TO_STRING(Rack_HMI.Rack_Cell_Pcalc.Field.BSA_Cell_MaxV_Location) ;

	HMI.BatteryInfo.BSA_Cell_MaxV_Location		:= CONCAT(HMI.BatteryInfo.BSA_Cell_MaxV_Cell_Location,'(C)');
	HMI.BatteryInfo.BSA_Cell_MinV_Cell_Location		:= UINT_TO_STRING(Rack_HMI.Rack_Cell_Pcalc.Field.BSA_Cell_MinV_Location) ;

	HMI.BatteryInfo.BSA_Cell_MinV_Location		:= CONCAT(HMI.BatteryInfo.BSA_Cell_MinV_Cell_Location,'(C)');
	HMI.BatteryInfo.BSA_Cell_MaxT_Cell_Location		:= UINT_TO_STRING((Rack_HMI.Rack_Cell_Pcalc.Field.BSA_Cell_MaxT_Location)) ;

	HMI.BatteryInfo.BSA_Cell_MaxT_Location		:= CONCAT(HMI.BatteryInfo.BSA_Cell_MaxT_Cell_Location,'(C)');

	HMI.BatteryInfo.BSA_Cell_MinT_Cell_Location 		:= UINT_TO_STRING(Rack_HMI.Rack_Cell_Pcalc.Field.BSA_Cell_MinT_Location) ;

	HMI.BatteryInfo.BSA_Cell_MinT_Location		:= CONCAT(HMI.BatteryInfo.BSA_Cell_MinT_Cell_Location,'(C)');

	HMI.Module1Info.Volt_Total_A 	:= REAL_TO_STRING(Rack_HMI.Modul1_Info.Field.Volt_Total) ;
	HMI.Module1Info.Volt_Total_B		:= CONCAT(HMI.Module1Info.Volt_Total_A,'(V)');

	IF (Rack_HMI.Modul1_Info.Field.OPS_Fault) THEN
		HMI.Module1Info.OPS_Fault := 'Solid_Red';
	ELSE
		HMI.Module1Info.OPS_Fault := 'Solid_Green';
	END_IF;

	IF (Rack_HMI.Modul1_Info.Field.OPS_MBCOM_Err) THEN
		HMI.Module1Info.OPS_MBCOM_Err := 'Solid_Red';
	ELSE
		HMI.Module1Info.OPS_MBCOM_Err := 'Solid_Green';
	END_IF;

	IF (Rack_HMI.Modul1_Info.Field.CTCOM_Err) THEN
		HMI.Module1Info.CTCOM_Err := 'Solid_Red';
	ELSE
		HMI.Module1Info.CTCOM_Err := 'Solid_Green';
	END_IF;

	HMI.Module2Info.Volt_Total_A 	:= REAL_TO_STRING(Rack_HMI.Modul2_Info.Field.Volt_Total) ;
	HMI.Module2Info.Volt_Total_B		:= CONCAT(HMI.Module2Info.Volt_Total_A,'(V)');

	IF (Rack_HMI.Modul2_Info.Field.OPS_Fault) THEN
		HMI.Module2Info.OPS_Fault := 'Solid_Red';
	ELSE
		HMI.Module2Info.OPS_Fault := 'Solid_Green';
	END_IF;

	IF (Rack_HMI.Modul2_Info.Field.OPS_MBCOM_Err) THEN
		HMI.Module2Info.OPS_MBCOM_Err := 'Solid_Red';
	ELSE
		HMI.Module2Info.OPS_MBCOM_Err := 'Solid_Green';
	END_IF;

	IF (Rack_HMI.Modul2_Info.Field.CTCOM_Err) THEN
		HMI.Module2Info.CTCOM_Err := 'Solid_Red';
	ELSE
		HMI.Module2Info.CTCOM_Err := 'Solid_Green';
	END_IF;

	HMI.Module3Info.Volt_Total_A 	:= REAL_TO_STRING(Rack_HMI.Modul3_Info.Field.Volt_Total) ;
	HMI.Module3Info.Volt_Total_B		:= CONCAT(HMI.Module3Info.Volt_Total_A,'(V)');

	IF (Rack_HMI.Modul3_Info.Field.OPS_Fault) THEN
		HMI.Module3Info.OPS_Fault := 'Solid_Red';
	ELSE
		HMI.Module3Info.OPS_Fault := 'Solid_Green';
	END_IF;

	IF (Rack_HMI.Modul3_Info.Field.OPS_MBCOM_Err) THEN
		HMI.Module3Info.OPS_MBCOM_Err := 'Solid_Red';
	ELSE
		HMI.Module3Info.OPS_MBCOM_Err := 'Solid_Green';
	END_IF;

	IF (Rack_HMI.Modul3_Info.Field.CTCOM_Err) THEN
		HMI.Module3Info.CTCOM_Err := 'Solid_Red';
	ELSE
		HMI.Module3Info.CTCOM_Err := 'Solid_Green';
	END_IF;

	HMI.Module4Info.Volt_Total_A 	:= REAL_TO_STRING(Rack_HMI.Modul4_Info.Field.Volt_Total) ;
	HMI.Module4Info.Volt_Total_B		:= CONCAT(HMI.Module4Info.Volt_Total_A,'(V)');

	IF (Rack_HMI.Modul4_Info.Field.OPS_Fault) THEN
		HMI.Module4Info.OPS_Fault := 'Solid_Red';
	ELSE
		HMI.Module4Info.OPS_Fault := 'Solid_Green';
	END_IF;

	IF (Rack_HMI.Modul4_Info.Field.OPS_MBCOM_Err) THEN
		HMI.Module4Info.OPS_MBCOM_Err := 'Solid_Red';
	ELSE
		HMI.Module4Info.OPS_MBCOM_Err := 'Solid_Green';
	END_IF;

	IF (Rack_HMI.Modul4_Info.Field.CTCOM_Err) THEN
		HMI.Module4Info.CTCOM_Err := 'Solid_Red';
	ELSE
		HMI.Module4Info.CTCOM_Err := 'Solid_Green';
	END_IF;

	HMI.Module5Info.Volt_Total_A 	:= REAL_TO_STRING(Rack_HMI.Modul5_Info.Field.Volt_Total) ;
	HMI.Module5Info.Volt_Total_B		:= CONCAT(HMI.Module5Info.Volt_Total_A,'(V)');

	IF (Rack_HMI.Modul5_Info.Field.OPS_Fault) THEN
		HMI.Module5Info.OPS_Fault := 'Solid_Red';
	ELSE
		HMI.Module5Info.OPS_Fault := 'Solid_Green';
	END_IF;

	IF (Rack_HMI.Modul5_Info.Field.OPS_MBCOM_Err) THEN
		HMI.Module5Info.OPS_MBCOM_Err := 'Solid_Red';
	ELSE
		HMI.Module5Info.OPS_MBCOM_Err := 'Solid_Green';
	END_IF;

	IF (Rack_HMI.Modul5_Info.Field.CTCOM_Err) THEN
		HMI.Module5Info.CTCOM_Err := 'Solid_Red';
	ELSE
		HMI.Module5Info.CTCOM_Err := 'Solid_Green';
	END_IF;

	HMI.Module6Info.Volt_Total_A 	:= REAL_TO_STRING(Rack_HMI.Modul6_Info.Field.Volt_Total) ;
	HMI.Module6Info.Volt_Total_B		:= CONCAT(HMI.Module6Info.Volt_Total_A,'(V)');

	IF (Rack_HMI.Modul6_Info.Field.OPS_Fault) THEN
		HMI.Module6Info.OPS_Fault := 'Solid_Red';
	ELSE
		HMI.Module6Info.OPS_Fault := 'Solid_Green';
	END_IF;

	IF (Rack_HMI.Modul6_Info.Field.OPS_MBCOM_Err) THEN
		HMI.Module6Info.OPS_MBCOM_Err := 'Solid_Red';
	ELSE
		HMI.Module6Info.OPS_MBCOM_Err := 'Solid_Green';
	END_IF;

	IF (Rack_HMI.Modul6_Info.Field.CTCOM_Err) THEN
		HMI.Module6Info.CTCOM_Err := 'Solid_Red';
	ELSE
		HMI.Module6Info.CTCOM_Err := 'Solid_Green';
	END_IF;

	HMI.Module7Info.Volt_Total_A 	:= REAL_TO_STRING(Rack_HMI.Modul7_Info.Field.Volt_Total) ;
	HMI.Module7Info.Volt_Total_B		:= CONCAT(HMI.Module7Info.Volt_Total_A,'(V)');

	IF (Rack_HMI.Modul7_Info.Field.OPS_Fault) THEN
		HMI.Module7Info.OPS_Fault := 'Solid_Red';
	ELSE
		HMI.Module7Info.OPS_Fault := 'Solid_Green';
	END_IF;

	IF (Rack_HMI.Modul7_Info.Field.OPS_MBCOM_Err) THEN
		HMI.Module7Info.OPS_MBCOM_Err := 'Solid_Red';
	ELSE
		HMI.Module7Info.OPS_MBCOM_Err := 'Solid_Green';
	END_IF;

	IF (Rack_HMI.Modul7_Info.Field.CTCOM_Err) THEN
		HMI.Module7Info.CTCOM_Err := 'Solid_Red';
	ELSE
		HMI.Module7Info.CTCOM_Err := 'Solid_Green';
	END_IF;

	IF Rack_HMI.Rack_State.Field.BSA_Water_leak THEN
		HMI.DIOStatus.BSA_Water_leak			:= 'Solid_Red';
	ELSE
		HMI.DIOStatus.BSA_Water_leak			:= 'Solid_Green';
	END_IF;
	IF Rack_HMI.Rack_State.Field.BSA_Neg_Rly THEN
		HMI.DIOStatus.BSA_Neg_Rly		:= 'Solid_Red';
	ELSE
		HMI.DIOStatus.BSA_Neg_Rly		:= 'Solid_Green';
	END_IF;
	IF Rack_HMI.Rack_State.Field.BSA_Pos_Rly THEN
		HMI.DIOStatus.BSA_Pos_Rly		:= 'Solid_Red';
	ELSE
		HMI.DIOStatus.BSA_Pos_Rly		:= 'Solid_Green';
	END_IF;
	IF Rack_HMI.Rack_State.Field.BSA_PreChar_Rly THEN
		HMI.DIOStatus.BSA_PreChar_Rly		:= 'Solid_Red';
	ELSE
		HMI.DIOStatus.BSA_PreChar_Rly		:= 'Solid_Green';
	END_IF;

	(* Over Current *)
	IF Rack_HMI.Rack_AlarmState.Field.protect.BSA_Prtct_Chager_OC  THEN
		HMI.ProtectStatus.BSA_Charge_OC		:= 'Solid_Red';
	ELSIF Rack_HMI.Rack_AlarmState.Field.fault.BSA_FLT_Chager_OC  THEN
		HMI.ProtectStatus.BSA_Charge_OC		:= 'Solid_Orange';
	ELSIF Rack_HMI.Rack_AlarmState.Field.warning.BSA_Wn_Chager_OC  THEN
		HMI.ProtectStatus.BSA_Charge_OC		:= 'Solid_Yellow';
	ELSE
		HMI.ProtectStatus.BSA_Charge_OC		:= 'Solid_Green';
	END_IF;
	IF Rack_HMI.Rack_AlarmState.Field.protect.BSA_Prtct_Dischager_OC THEN
		HMI.ProtectStatus.BSA_Discharge_OC		:= 'Solid_Red';
	ELSIF  Rack_HMI.Rack_AlarmState.Field.fault.BSA_FLT_Dischager_OC THEN
		HMI.ProtectStatus.BSA_Discharge_OC		:= 'Solid_Orange';
	ELSIF Rack_HMI.Rack_AlarmState.Field.warning.BSA_Wn_Dischager_OC THEN
		HMI.ProtectStatus.BSA_Discharge_OC		:= 'Solid_Yellow';
	ELSE
		HMI.ProtectStatus.BSA_Discharge_OC		:= 'Solid_Green';
	END_IF;

	IF Rack_HMI.Rack_AlarmState.Field.protect.BSA_Prtct_SOC_OV THEN
		HMI.ProtectStatus.BSA_SOC_OV		:= 'Solid_Red';
	ELSIF Rack_HMI.Rack_AlarmState.Field.fault.BSA_FLT_SOC_OV THEN
		HMI.ProtectStatus.BSA_SOC_OV		:= 'Solid_Orange';
	ELSIF Rack_HMI.Rack_AlarmState.Field.warning.BSA_Wn_SOC_OV THEN
		HMI.ProtectStatus.BSA_SOC_OV		:= 'Solid_Yellow';
	ELSE
		HMI.ProtectStatus.BSA_SOC_OV		:= 'Solid_Green';
	END_IF;

	IF Rack_HMI.Rack_AlarmState.Field.protect.BSA_Prtct_SOC_Un THEN
		HMI.ProtectStatus.BSA_SOC_Un		:= 'Solid_Red';
	ELSIF Rack_HMI.Rack_AlarmState.Field.fault.BSA_FLT_SOC_Un THEN
		HMI.ProtectStatus.BSA_SOC_Un		:= 'Solid_Orange';
	ELSIF Rack_HMI.Rack_AlarmState.Field.warning.BSA_Wn_SOC_Un THEN
		HMI.ProtectStatus.BSA_SOC_Un		:= 'Solid_Yellow';
	ELSE
		HMI.ProtectStatus.BSA_SOC_Un		:= 'Solid_Green';
	END_IF;

	IF Rack_HMI.Rack_AlarmState.Field.protect.BSA_Prtct_OV THEN
		HMI.ProtectStatus.BSA_OV		:= 'Solid_Red';
	ELSIF Rack_HMI.Rack_AlarmState.Field.fault.BSA_FLT_OV THEN
		HMI.ProtectStatus.BSA_OV		:= 'Solid_Orange';
	ELSIF Rack_HMI.Rack_AlarmState.Field.warning.BSA_Wn_OV THEN
		HMI.ProtectStatus.BSA_OV		:= 'Solid_Yellow';
	ELSE
		HMI.ProtectStatus.BSA_OV		:= 'Solid_Green';
	END_IF;

	IF Rack_HMI.Rack_AlarmState.Field.protect.BSA_Prtct_UV THEN
		HMI.ProtectStatus.BSA_UV		:= 'Solid_Red';
	ELSIF Rack_HMI.Rack_AlarmState.Field.fault.BSA_FLT_UV THEN
		HMI.ProtectStatus.BSA_UV		:= 'Solid_Orange';
	ELSIF Rack_HMI.Rack_AlarmState.Field.warning.BSA_Wn_UV  THEN
		HMI.ProtectStatus.BSA_UV		:= 'Solid_Yellow';
	ELSE
		HMI.ProtectStatus.BSA_UV		:= 'Solid_Green';
	END_IF;

	IF Rack_HMI.Rack_AlarmState.Field.protect.BSA_Prtct_Cell_OV THEN
		HMI.ProtectStatus.BSA_Cell_OV		:= 'Solid_Red';
	ELSIF Rack_HMI.Rack_AlarmState.Field.fault.BSA_FLT_Cell_OV THEN
		HMI.ProtectStatus.BSA_Cell_OV		:= 'Solid_Orange';
	ELSIF Rack_HMI.Rack_AlarmState.Field.warning.BSA_Wn_Cell_OV THEN
		HMI.ProtectStatus.BSA_Cell_OV		:= 'Solid_Yellow';
	ELSE
		HMI.ProtectStatus.BSA_Cell_OV		:= 'Solid_Green';
	END_IF;

	IF Rack_HMI.Rack_AlarmState.Field.protect.BSA_Prtct_Cell_UV THEN
		HMI.ProtectStatus.BSA_Cell_UV		:= 'Solid_Red';
	ELSIF Rack_HMI.Rack_AlarmState.Field.fault.BSA_FLT_Cell_UV THEN
		HMI.ProtectStatus.BSA_Cell_UV		:= 'Solid_Orange';
	ELSIF Rack_HMI.Rack_AlarmState.Field.warning.BSA_Wn_Cell_UV THEN
		HMI.ProtectStatus.BSA_Cell_UV		:= 'Solid_Yellow';
	ELSE
		HMI.ProtectStatus.BSA_Cell_UV		:= 'Solid_Green';
	END_IF;

	IF Rack_HMI.Rack_AlarmState.Field.protect.BSA_Prtct_Cell_UnbalV THEN
		HMI.ProtectStatus.BSA_Cell_UnbalV		:= 'Solid_Red';
	ELSIF Rack_HMI.Rack_AlarmState.Field.fault.BSA_FLT_Cell_UnbalV THEN
		HMI.ProtectStatus.BSA_Cell_UnbalV		:= 'Solid_Orange';
	ELSIF Rack_HMI.Rack_AlarmState.Field.warning.BSA_Wn_Cell_UnbalV THEN
		HMI.ProtectStatus.BSA_Cell_UnbalV		:= 'Solid_Yellow';
	ELSE
		HMI.ProtectStatus.BSA_Cell_UnbalV		:= 'Solid_Green';
	END_IF;

	IF Rack_HMI.Rack_AlarmState.Field.protect.BSA_Prtct_DisCharger_Cell_OT THEN
		HMI.ProtectStatus.BSA_DisCharger_Cell_OT		:= 'Solid_Red';
	ELSIF Rack_HMI.Rack_AlarmState.Field.fault.BSA_FLT_DisCharger_Cell_OT THEN
		HMI.ProtectStatus.BSA_DisCharger_Cell_OT		:= 'Solid_Orange';
	ELSIF Rack_HMI.Rack_AlarmState.Field.warning.BSA_Wn_DisCharger_Cell_OT THEN
		HMI.ProtectStatus.BSA_DisCharger_Cell_OT		:= 'Solid_Yellow';
	ELSE
		HMI.ProtectStatus.BSA_DisCharger_Cell_OT		:= 'Solid_Green';
	END_IF;

	IF Rack_HMI.Rack_AlarmState.Field.protect.BSA_Prtct_Charger_Cell_OT THEN
		HMI.ProtectStatus.BSA_Charger_Cell_OT		:= 'Solid_Red';
	ELSIF Rack_HMI.Rack_AlarmState.Field.fault.BSA_FLT_Charger_Cell_OT THEN
		HMI.ProtectStatus.BSA_Charger_Cell_OT		:= 'Solid_Orange';
	ELSIF Rack_HMI.Rack_AlarmState.Field.warning.BSA_Wn_Charger_Cell_OT THEN
		HMI.ProtectStatus.BSA_Charger_Cell_OT		:= 'Solid_Yellow';
	ELSE
		HMI.ProtectStatus.BSA_Charger_Cell_OT		:= 'Solid_Green';
	END_IF;

	IF Rack_HMI.Rack_AlarmState.Field.protect.BSA_Prtct_DisCharger_Cell_UT THEN
		HMI.ProtectStatus.BSA_DisCharger_Cell_UT		:= 'Solid_Red';
	ELSIF Rack_HMI.Rack_AlarmState.Field.fault.BSA_FLT_DisCharger_Cell_UT THEN
		HMI.ProtectStatus.BSA_DisCharger_Cell_UT		:= 'Solid_Orange';
	ELSIF Rack_HMI.Rack_AlarmState.Field.warning.BSA_Wn_DisCharger_Cell_UT THEN
		HMI.ProtectStatus.BSA_DisCharger_Cell_UT		:= 'Solid_Yellow';
	ELSE
		HMI.ProtectStatus.BSA_DisCharger_Cell_UT		:= 'Solid_Green';
	END_IF;

	IF Rack_HMI.Rack_AlarmState.Field.protect.BSA_Prtct_Charger_Cell_UT THEN
		HMI.ProtectStatus.BSA_Charger_Cell_UT		:= 'Solid_Red';
	ELSIF Rack_HMI.Rack_AlarmState.Field.fault.BSA_FLT_Charger_Cell_UT THEN
		HMI.ProtectStatus.BSA_Charger_Cell_UT		:= 'Solid_Orange';
	ELSIF Rack_HMI.Rack_AlarmState.Field.warning.BSA_Wn_Charger_Cell_UT THEN
		HMI.ProtectStatus.BSA_Charger_Cell_UT		:= 'Solid_Yellow';
	ELSE
		HMI.ProtectStatus.BSA_Charger_Cell_UT		:= 'Solid_Green';
	END_IF;

	IF Rack_HMI.Rack_AlarmState.Field.protect.BSA_Prtct_Cell_UnbalT THEN
		HMI.ProtectStatus.BSA_Cell_UnbalT			:= 'Solid_Red';
	ELSIF Rack_HMI.Rack_AlarmState.Field.fault.BSA_FLT_Cell_UnbalT THEN
		HMI.ProtectStatus.BSA_Cell_UnbalT			:= 'Solid_Orange';
	ELSIF Rack_HMI.Rack_AlarmState.Field.warning.BSA_Wn_Cell_UnbalT THEN
		HMI.ProtectStatus.BSA_Cell_UnbalT			:= 'Solid_Yellow';
	ELSE
		HMI.ProtectStatus.BSA_Cell_UnbalT			:= 'Solid_Green';
	END_IF;

	IF Rack_HMI.Rack_AlarmState.Field.protect.BSA_Prtct_Discharger_UnbaPWR THEN
		HMI.ProtectStatus.BSA_Discharge_Unbal_PWR	:= 'Solid_Red';
	ELSIF Rack_HMI.Rack_AlarmState.Field.fault.BSA_FLT_Discharger_UnbaPWR THEN
		HMI.ProtectStatus.BSA_Discharge_Unbal_PWR	:= 'Solid_Orange';
	ELSIF Rack_HMI.Rack_AlarmState.Field.warning.BSA_Wn_Discharger_UnbaPWR THEN
		HMI.ProtectStatus.BSA_Discharge_Unbal_PWR	:= 'Solid_Yellow';
	ELSE
		HMI.ProtectStatus.BSA_Discharge_Unbal_PWR	:= 'Solid_Green';
	END_IF;

	IF Rack_HMI.Rack_AlarmState.Field.protect.BSA_Prtct_Charger_UnbaPWR THEN
		HMI.ProtectStatus.BSA_Charge_Unbal_PWR		:= 'Solid_Red';
	ELSIF Rack_HMI.Rack_AlarmState.Field.fault.BSA_FLT_Charger_UnbaPWR THEN
		HMI.ProtectStatus.BSA_Charge_Unbal_PWR		:= 'Solid_Orange';
	ELSIF Rack_HMI.Rack_AlarmState.Field.warning.BSA_Wn_Charger_UnbaPWR THEN
		HMI.ProtectStatus.BSA_Charge_Unbal_PWR		:= 'Solid_Yellow';
	ELSE
		HMI.ProtectStatus.BSA_Charge_Unbal_PWR		:= 'Solid_Green';
	END_IF;

	IF Rack_HMI.Rack_AlarmState.Field.protect.BSA_Prtct_Rly_Err THEN
		HMI.ProtectStatus.BSA_Prtct_Rly_Err			:= 'Solid_Red';
	ELSE
		HMI.ProtectStatus.BSA_Prtct_Rly_Err			:= 'Solid_Green';
	END_IF;
	IF Rack_HMI.Rack_AlarmState.Field.protect.BSA_Prtct_IN_COM_Err THEN
		HMI.ProtectStatus.BSA_Prtct_IN_COM_Err		:= 'Solid_Red';
	ELSE
		HMI.ProtectStatus.BSA_Prtct_IN_COM_Err		:= 'Solid_Green';
	END_IF;
	IF Rack_HMI.Rack_AlarmState.Field.protect.BSA_Prtct_EX_COM_Err THEN
		HMI.ProtectStatus.BSA_Prtct_EX_COM_Err		:= 'Solid_Red';
	ELSE
		HMI.ProtectStatus.BSA_Prtct_EX_COM_Err		:= 'Solid_Green';
	END_IF;
	//	IF Rack_HMI.Rack_AlarmState.Field.protect.BSA_Prtct_CT_COM_Err THEN
	//		HMI.ProtectStatus.BSA_Prtct_InsulationRegister		:= 'Solid_Red';
	//	ELSE
	//		HMI.ProtectStatus.BSA_Prtct_InsulationRegister		:= 'Solid_Green';
	//	END_IF;
	IF Rack_HMI.Rack_AlarmState.Field.protect.BSA_Prtct_Water_Leak_Err THEN
		HMI.ProtectStatus.BSA_Prtct_Water_Leak_Err	:= 'Solid_Red';
	ELSE
		HMI.ProtectStatus.BSA_Prtct_Water_Leak_Err	:= 'Solid_Green';
	END_IF;
	//	IF Rack_HMI.Rack_AlarmState.Field.protect.BSA_Prtct_EMS_SW_Err THEN
	//		HMI.ProtectStatus.BSA_Prtct_MDS		:= 'Solid_Red';
	//	ELSE
	//		HMI.ProtectStatus.BSA_Prtct_MDS		:= 'Solid_Green';
	//	END_IF;

	(* DIO *)
	//	IF HMI.Rack1[19].0 THEN
	//		HMIBinding.RackUI.sString20[34] 		:= 'Solid_Red';
	//	ELSE
	//		HMIBinding.RackUI.sString20[34]			:= 'Solid_Green';
	//	END_IF;
	//	IF HMI.Rack1[19].1 THEN
	//		HMIBinding.RackUI.sString20[35] 		:= 'Solid_Red';
	//	ELSE
	//		HMIBinding.RackUI.sString20[35]			:= 'Solid_Green';
	//	END_IF;
	//	IF HMI.Rack1[19].2 THEN
	//		HMIBinding.RackUI.sString20[36] 		:= 'Solid_Red';
	//	ELSE
	//		HMIBinding.RackUI.sString20[36]			:= 'Solid_Green';
	//	END_IF;
	//	IF HMI.Rack1[20].2 THEN
	//		HMIBinding.RackUI.sString20[37] 		:= 'Solid_Red';
	//	ELSE
	//		HMIBinding.RackUI.sString20[37]			:= 'Solid_Green';
	//	END_IF;
	//	IF HMI.Rack1[20].4 THEN
	//		HMIBinding.RackUI.sString20[38] 		:= 'Solid_Red';
	//	ELSE
	//		HMIBinding.RackUI.sString20[38]			:= 'Solid_Green';
	//	END_IF;
	//	IF HMI.Rack1[20].5 THEN
	//		HMIBinding.RackUI.sString20[39] 		:= 'Solid_Red';
	//	ELSE
	//		HMIBinding.RackUI.sString20[39]			:= 'Solid_Green';
	//	END_IF;

END_ACTION
```

#### HMI_System.st
```iecst
ACTION AtSystemUI :

	CASE System_HMI.SysBatCal.Field.BSA_Divice_Status OF
		0:  HMI.BSA_Divice_Status := 'INIT';
		1:  HMI.BSA_Divice_Status := 'READY';
		2:  HMI.BSA_Divice_Status := 'STANDBY';
		3:  HMI.BSA_Divice_Status := 'RUN';
		4:  HMI.BSA_Divice_Status := 'PROTECT';
		5:  HMI.BSA_Divice_Status := 'STOP';
	END_CASE;

	HMI.Gauge.BRA_Volt_Total		:= (System_HMI.SysBatCal.Field.BSA_Volt_Total) ;
	HMI.Gauge.BRA_Volt_Total_A		:= REAL_TO_STRING((HMI.Gauge.BRA_Volt_Total-400)*0.675);
	HMI.Gauge.BRA_Volt_Total_B		:= CONCAT('[{"select":"#gauge3","spin":[',CONCAT(HMI.Gauge.BRA_Volt_Total_A,',0,0]}]'));

	HMI.Gauge.BRA_Curr_Total 			:= (System_HMI.SysBatCal.Field.BSA_Curr_Total) ;
	HMI.Gauge.BRA_Curr_Total_A		:= REAL_TO_STRING(HMI.Gauge.BRA_Curr_Total*0.27+135);
	HMI.Gauge.BRA_Curr_Total_B		:= CONCAT('[{"select":"#gauge4","spin":[',CONCAT(HMI.Gauge.BRA_Curr_Total_A,',0,0]}]'));

	HMI.Gauge.BRA_SOC		:= (System_HMI.SysBatCal.Field.BSA_SOC) ;
	HMI.Gauge.BRA_SOC_A		:= REAL_TO_STRING(HMI.Gauge.BRA_SOC*2.7);
	HMI.Gauge.BRA_SOC_B		:= CONCAT('[{"select":"#gauge1","spin":[',CONCAT(HMI.Gauge.BRA_SOC_A,',0,0]}]'));

	HMI.Gauge.BRA_SOH		:= (System_HMI.SysBatDIO.Field.BSA_SOH);
	HMI.Gauge.BRA_SOH_A		:= REAL_TO_STRING(HMI.Gauge.BRA_SOH*2.7);
	HMI.Gauge.BRA_SOH_B		:= CONCAT('[{"select":"#gauge2","spin":[',CONCAT(HMI.Gauge.BRA_SOH_A,',0,0]}]'));

	HMI.BatteryInfo.BSA_Cell_MaxV 		:= (System_HMI.SysCellVolt.Field.BSA_Cell_MaxV) ;
	HMI.BatteryInfo.BSA_Cell_MinV		:= (System_HMI.SysCellVolt.Field.BSA_Cell_MinV);
	HMI.BatteryInfo.BSA_Cell_AVGV		:= (System_HMI.SysCellVolt.Field.BSA_Cell_AVGV)  ;
	HMI.BatteryInfo.BSA_Cell_DeviV 		:= (System_HMI.SysCellVolt.Field.BSA_Cell_DeviV) ;

	HMI.BatteryInfo.BSA_Cell_MaxT 		:= (System_HMI.SysCellTemps.Field.BSA_Cell_MaxT) ;
	HMI.BatteryInfo.BSA_Cell_MinT		:= (System_HMI.SysCellTemps.Field.BSA_Cell_MinT	) ;
	HMI.BatteryInfo.BSA_Cell_AVGT		:= (System_HMI.SysCellTemps.Field.BSA_Cell_AVGT) ;
	HMI.BatteryInfo.BSA_Cell_DeviT 		:= (System_HMI.SysCellTemps.Field.BSA_Cell_DeviT);

	HMI.BatteryInfo.BSA_Cell_MaxV_Rack_Location		:= UINT_TO_STRING(System_HMI.SysCellV_TPos.Field.BSA_Rack_MaxV_Location) ;
	HMI.BatteryInfo.BSA_Cell_MaxV_Cell_Location		:= UINT_TO_STRING(System_HMI.SysCellV_TPos.Field.BSA_Cell_MaxV_Location) ;
	HMI.BatteryInfo.BSA_Cell_MaxV_Location		:= CONCAT(HMI.BatteryInfo.BSA_Cell_MaxV_Rack_Location,CONCAT('(R), ',CONCAT(HMI.BatteryInfo.BSA_Cell_MaxV_Cell_Location,'(C)')));

	HMI.BatteryInfo.BSA_Cell_MinV_Rack_Location		:= UINT_TO_STRING(System_HMI.SysCellV_TPos.Field.BSA_Rack_MinV_Location) ;
	HMI.BatteryInfo.BSA_Cell_MinV_Cell_Location		:= UINT_TO_STRING(System_HMI.SysCellV_TPos.Field.BSA_Cell_MinV_Location) ;
	HMI.BatteryInfo.BSA_Cell_MinV_Location		:= CONCAT(HMI.BatteryInfo.BSA_Cell_MinV_Rack_Location,CONCAT('(R), ',CONCAT(HMI.BatteryInfo.BSA_Cell_MinV_Cell_Location,'(C)')));

	HMI.BatteryInfo.BSA_Cell_MaxT_Rack_Location		:= UINT_TO_STRING(System_HMI.SysCellV_TPos.Field.BSA_Rack_MaxT_Location) ;
	HMI.BatteryInfo.BSA_Cell_MaxT_Cell_Location		:= UINT_TO_STRING(System_HMI.SysCellV_TPos.Field.BSA_Cell_MaxT_Location) ;
	HMI.BatteryInfo.BSA_Cell_MaxT_Location		:= CONCAT(HMI.BatteryInfo.BSA_Cell_MaxT_Rack_Location,CONCAT('(R), ',CONCAT(HMI.BatteryInfo.BSA_Cell_MaxT_Cell_Location,'(C)')));

	HMI.BatteryInfo.BSA_Cell_MinT_Rack_Location		:= UINT_TO_STRING(System_HMI.SysCellV_TPos.Field.BSA_Rack_MinT_Location) ;
	HMI.BatteryInfo.BSA_Cell_MinT_Cell_Location		:= UINT_TO_STRING(System_HMI.SysCellV_TPos.Field.BSA_Cell_MinT_Location) ;
	HMI.BatteryInfo.BSA_Cell_MinT_Location		:= CONCAT(HMI.BatteryInfo.BSA_Cell_MinT_Rack_Location,CONCAT('(R), ',CONCAT(HMI.BatteryInfo.BSA_Cell_MinT_Cell_Location,'(C)')));

	IF System_HMI.SysBatProtect.Field.BSA_Prtct_WaterLeak THEN
		HMI.DIOStatus.BSA_Water_leak	:= 'Solid_Red';
	ELSE
		HMI.DIOStatus.BSA_Water_leak	:= 'Solid_Green';
	END_IF;

	IF System_HMI.SysBatDIO.Field.BSA_Prelay_DO_Status THEN
		HMI.DIOStatus.BSA_Neg_Rly		:= 'Solid_Red';
	ELSE
		HMI.DIOStatus.BSA_Neg_Rly		:= 'Solid_Green';
	END_IF;
	IF System_HMI.SysBatDIO.Field.BSA_Nrelay_DO_Status THEN
		HMI.DIOStatus.BSA_Pos_Rly		:= 'Solid_Red';
	ELSE
		HMI.DIOStatus.BSA_Pos_Rly		:= 'Solid_Green';
	END_IF;
	IF System_HMI.SysBatDIO.Field.BSA_ProRelay_DO_Status THEN
		HMI.DIOStatus.BSA_PreChar_Rly	:= 'Solid_Red';
	ELSE
		HMI.DIOStatus.BSA_PreChar_Rly	:= 'Solid_Green';
	END_IF;

	IF System_HMI.SysBatProtect.Field.BSA_Prtct_OC THEN
		HMI.ProtectStatus.BSA_OC		:= 'Solid_Red';
	ELSIF System_HMI.SysBatProtect.Field.BSA_Fault_OC THEN
		HMI.ProtectStatus.BSA_OC		:= 'Solid_Orange';
	ELSIF System_HMI.SysBatProtect.Field.BSA_Alarm_OC THEN
		HMI.ProtectStatus.BSA_OC		:= 'Solid_Yellow';
	ELSE
		HMI.ProtectStatus.BSA_OC		:= 'Solid_Green';
	END_IF;

	IF System_HMI.SysBatProtect.Field.BSA_Prtct_SOC_OV THEN
		HMI.ProtectStatus.BSA_SOC_OV		:= 'Solid_Red';
	ELSIF System_HMI.SysBatProtect.Field.BSA_Fault_SOC_OV THEN
		HMI.ProtectStatus.BSA_SOC_OV		:= 'Solid_Orange';
	ELSIF System_HMI.SysBatProtect.Field.BSA_Alarm_SOC_OV THEN
		HMI.ProtectStatus.BSA_SOC_OV		:= 'Solid_Yellow';
	ELSE
		HMI.ProtectStatus.BSA_SOC_OV		:= 'Solid_Green';
	END_IF;

	IF System_HMI.SysBatProtect.Field.BSA_Prtct_SOC_UN THEN
		HMI.ProtectStatus.BSA_SOC_Un		:= 'Solid_Red';
	ELSIF System_HMI.SysBatProtect.Field.BSA_Fault_SOC_UN THEN
		HMI.ProtectStatus.BSA_SOC_Un		:= 'Solid_Orange';
	ELSIF System_HMI.SysBatProtect.Field.BSA_Alarm_SOC_UN THEN
		HMI.ProtectStatus.BSA_SOC_Un		:= 'Solid_Yellow';
	ELSE
		HMI.ProtectStatus.BSA_SOC_Un		:= 'Solid_Green';
	END_IF;

	IF System_HMI.SysBatProtect.Field.BSA_Prtct_OV THEN
		HMI.ProtectStatus.BSA_OV		:= 'Solid_Red';
	ELSIF System_HMI.SysBatProtect.Field.BSA_Fault_OV THEN
		HMI.ProtectStatus.BSA_OV		:= 'Solid_Orange';
	ELSIF System_HMI.SysBatProtect.Field.BSA_Alarm_OV THEN
		HMI.ProtectStatus.BSA_OV		:= 'Solid_Yellow';
	ELSE
		HMI.ProtectStatus.BSA_OV		:= 'Solid_Green';
	END_IF;

	IF System_HMI.SysBatProtect.Field.BSA_Prtct_UV THEN
		HMI.ProtectStatus.BSA_UV		:= 'Solid_Red';
	ELSIF System_HMI.SysBatProtect.Field.BSA_Fault_UV THEN
		HMI.ProtectStatus.BSA_UV		:= 'Solid_Orange';
	ELSIF System_HMI.SysBatProtect.Field.BSA_Alarm_UV  THEN
		HMI.ProtectStatus.BSA_UV		:= 'Solid_Yellow';
	ELSE
		HMI.ProtectStatus.BSA_UV		:= 'Solid_Green';
	END_IF;

	IF System_HMI.SysBatProtect.Field.BSA_Prtct_Cell_OV THEN
		HMI.ProtectStatus.BSA_Cell_OV		:= 'Solid_Red';
	ELSIF System_HMI.SysBatProtect.Field.BSA_Fault_Cell_OV THEN
		HMI.ProtectStatus.BSA_Cell_OV		:= 'Solid_Orange';
	ELSIF System_HMI.SysBatProtect.Field.BSA_Alarm_Cell_OV THEN
		HMI.ProtectStatus.BSA_Cell_OV		:= 'Solid_Yellow';
	ELSE
		HMI.ProtectStatus.BSA_Cell_OV		:= 'Solid_Green';
	END_IF;

	IF System_HMI.SysBatProtect.Field.BSA_Prtct_Cell_UV THEN
		HMI.ProtectStatus.BSA_Cell_UV		:= 'Solid_Red';
	ELSIF System_HMI.SysBatProtect.Field.BSA_Fault_Cell_UV THEN
		HMI.ProtectStatus.BSA_Cell_UV		:= 'Solid_Orange';
	ELSIF System_HMI.SysBatProtect.Field.BSA_Alarm_Cell_UV THEN
		HMI.ProtectStatus.BSA_Cell_UV		:= 'Solid_Yellow';
	ELSE
		HMI.ProtectStatus.BSA_Cell_UV		:= 'Solid_Green';
	END_IF;

	IF System_HMI.SysBatProtect.Field.BSA_Prtct_Cell_UnBalaV THEN
		HMI.ProtectStatus.BSA_Cell_UnbalV		:= 'Solid_Red';
	ELSIF System_HMI.SysBatProtect.Field.BSA_Fault_Cell_UnBalaV THEN
		HMI.ProtectStatus.BSA_Cell_UnbalV		:= 'Solid_Orange';
	ELSIF System_HMI.SysBatProtect.Field.BSA_Alarm_Cell_UnBalaV THEN
		HMI.ProtectStatus.BSA_Cell_UnbalV		:= 'Solid_Yellow';
	ELSE
		HMI.ProtectStatus.BSA_Cell_UnbalV		:= 'Solid_Green';
	END_IF;

	IF System_HMI.SysBatProtect.Field.BSA_Prtct_Discharger_Cell_OT THEN
		HMI.ProtectStatus.BSA_DisCharger_Cell_OT		:= 'Solid_Red';
	ELSIF System_HMI.SysBatProtect.Field.BSA_Fault_Discharger_Cell_OT THEN
		HMI.ProtectStatus.BSA_DisCharger_Cell_OT		:= 'Solid_Orange';
	ELSIF System_HMI.SysBatProtect.Field.BSA_Alarm_Discharger_Cell_OT THEN
		HMI.ProtectStatus.BSA_DisCharger_Cell_OT		:= 'Solid_Yellow';
	ELSE
		HMI.ProtectStatus.BSA_DisCharger_Cell_OT		:= 'Solid_Green';
	END_IF;

	IF System_HMI.SysBatProtect.Field.BSA_Prtct_Charger_Cell_OT THEN
		HMI.ProtectStatus.BSA_Charger_Cell_OT		:= 'Solid_Red';
	ELSIF System_HMI.SysBatProtect.Field.BSA_Fault_Charger_Cell_OT THEN
		HMI.ProtectStatus.BSA_Charger_Cell_OT		:= 'Solid_Orange';
	ELSIF System_HMI.SysBatProtect.Field.BSA_Alarm_Charger_Cell_OT THEN
		HMI.ProtectStatus.BSA_Charger_Cell_OT		:= 'Solid_Yellow';
	ELSE
		HMI.ProtectStatus.BSA_Charger_Cell_OT		:= 'Solid_Green';
	END_IF;

	IF System_HMI.SysBatProtect.Field.BSA_Prtct_Discharger_Cell_OT THEN
		HMI.ProtectStatus.BSA_DisCharger_Cell_UT		:= 'Solid_Red';
	ELSIF System_HMI.SysBatProtect.Field.BSA_Fault_Discharger_Cell_UT THEN
		HMI.ProtectStatus.BSA_DisCharger_Cell_UT		:= 'Solid_Orange';
	ELSIF System_HMI.SysBatProtect.Field.BSA_Alarm_Discharger_Cell_UT THEN
		HMI.ProtectStatus.BSA_DisCharger_Cell_UT		:= 'Solid_Yellow';
	ELSE
		HMI.ProtectStatus.BSA_DisCharger_Cell_UT		:= 'Solid_Green';
	END_IF;

	IF System_HMI.SysBatProtect.Field.BSA_Prtct_Discharger_Cell_UT THEN
		HMI.ProtectStatus.BSA_DisCharger_Cell_UT		:= 'Solid_Red';
	ELSIF System_HMI.SysBatProtect.Field.BSA_Fault_Discharger_Cell_UT THEN
		HMI.ProtectStatus.BSA_DisCharger_Cell_UT		:= 'Solid_Orange';
	ELSIF System_HMI.SysBatProtect.Field.BSA_Alarm_Discharger_Cell_UT THEN
		HMI.ProtectStatus.BSA_DisCharger_Cell_UT		:= 'Solid_Yellow';
	ELSE
		HMI.ProtectStatus.BSA_DisCharger_Cell_UT		:= 'Solid_Green';
	END_IF;

	IF System_HMI.SysBatProtect.Field.BSA_Prtct_Charger_Cell_UT THEN
		HMI.ProtectStatus.BSA_Charger_Cell_UT		:= 'Solid_Red';
	ELSIF System_HMI.SysBatProtect.Field.BSA_Fault_Charger_Cell_UT THEN
		HMI.ProtectStatus.BSA_Charger_Cell_UT		:= 'Solid_Orange';
	ELSIF System_HMI.SysBatProtect.Field.BSA_Alarm_Charger_Cell_UT THEN
		HMI.ProtectStatus.BSA_Charger_Cell_UT		:= 'Solid_Yellow';
	ELSE
		HMI.ProtectStatus.BSA_Charger_Cell_UT		:= 'Solid_Green';
	END_IF;

	IF System_HMI.SysBatProtect.Field.BSA_Prtct_Cell_UnBalaT THEN
		HMI.ProtectStatus.BSA_Cell_UnbalT		:= 'Solid_Red';
	ELSIF System_HMI.SysBatProtect.Field.BSA_Fault_Cell_UnBalaT THEN
		HMI.ProtectStatus.BSA_Cell_UnbalT		:= 'Solid_Orange';
	ELSIF System_HMI.SysBatProtect.Field.BSA_Alarm_Cell_UnBalaT THEN
		HMI.ProtectStatus.BSA_Cell_UnbalT		:= 'Solid_Yellow';
	ELSE
		HMI.ProtectStatus.BSA_Cell_UnbalT		:= 'Solid_Green';
	END_IF;

	IF System_HMI.SysBatProtect.Field.BSA_Prtct_InternalCOM THEN
		HMI.ProtectStatus.BSA_Prtct_IN_COM_Err		:= 'Solid_Red';
	ELSE
		HMI.ProtectStatus.BSA_Prtct_IN_COM_Err		:= 'Solid_Green';
	END_IF;
	IF System_HMI.SysBatProtect.Field.BSA_Prtct_ExternalCOM THEN
		HMI.ProtectStatus.BSA_Prtct_EX_COM_Err		:= 'Solid_Red';
	ELSE
		HMI.ProtectStatus.BSA_Prtct_EX_COM_Err		:= 'Solid_Green';
	END_IF;
	IF System_HMI.SysBatProtect.Field.BSA_Prtct_RelayWelding THEN
		HMI.ProtectStatus.BSA_Prtct_Rly_Err			:= 'Solid_Red';
	ELSE
		HMI.ProtectStatus.BSA_Prtct_Rly_Err			:= 'Solid_Green';
	END_IF;
	IF System_HMI.SysBatProtect.Field.BSA_Prtct_WaterLeak THEN
		HMI.ProtectStatus.BSA_Prtct_Water_Leak_Err	:= 'Solid_Red';
	ELSE
		HMI.ProtectStatus.BSA_Prtct_Water_Leak_Err	:= 'Solid_Green';
	END_IF;
	IF System_HMI.SysBatProtect.Field.BSA_Prtct_InsulationReg THEN
		HMI.ProtectStatus.BRA_Prtct_InsulationReg	:= 'Solid_Red';
	ELSE
		HMI.ProtectStatus.BRA_Prtct_InsulationReg	:= 'Solid_Green';
	END_IF;
	IF System_HMI.SysBatProtect.Field.BSA_Prtct_MDSFuse THEN
		HMI.ProtectStatus.BRA_Prtct_MDSFuse	:= 'Solid_Red';
	ELSE
		HMI.ProtectStatus.BRA_Prtct_MDSFuse	:= 'Solid_Green';
	END_IF;
	IF System_HMI.SysBatProtect.Field.BSA_Prtct_Cooling_System THEN
		HMI.ProtectStatus.BSA_Prtct_CoolingSystem		:= 'Solid_Red';
	ELSE
		HMI.ProtectStatus.BSA_Prtct_CoolingSystem		:= 'Solid_Green';
	END_IF;
END_ACTION
```
